// TIA Portal V16 program export: 10 tag tables, 22 data types, 19 data blocks, 13 code blocks (in call order from the OBs), 5 instance data blocks

VAR_GLOBAL   // PLC tag table "Default tag table"
END_VAR

VAR_GLOBAL   // PLC tag table "FC11001_Test"
   V001_FBK_OPEN AT %M100.0 : Bool;   // V001 Open limit switch
   V001_FBK_CLOSED AT %M100.1 : Bool;   // V001 Closed limit switch
   V001_FAULT AT %M100.2 : Bool;   // V001 External fault signal
   V001_OPERATE AT %M101.0 : Bool;   // V001 Energise (operate) signal
   V001_ESTOP AT %M100.3 : Bool;   // V001 Safety signal
   V001_TRIP AT %M100.4 : Bool;   // V001 Trip (interlock) signal
   V001_ILOCK AT %M100.5 : Bool;   // V001 Interlock signal
   V001_PERM AT %M100.6 : Bool;   // V001 Permissive (interlock) signal
   OpTimeRem AT %MD110 : Real;   // Operating timer last non-zero value
END_VAR

VAR_GLOBAL   // PLC tag table "FC19511_Test"
   SIM001_TRIGGER AT %M900.0 : Bool;   // Simulation Trigger Signal
   SIM001_OUTPUT AT %MD910 : Real;   // Simulation Output
   SIM001_INPUT AT %MD902 : Real;   // Simulation Input
   SIM001_Type AT %MW906 : Int;   // 0 = Step, 1 = Ramp, 2 = Sinusoid
   "Counter" AT %MW908 : Int;   // 100ms Counter
END_VAR

VAR_GLOBAL   // PLC tag table "FC19512"
   SIM001_TRIGGER AT %M900.0 : Bool;   // Simulation Trigger Signal
   SIM001_OUTPUT AT %MD910 : Real;
   SIM001_INPUT AT %MD902 : Real;
END_VAR

VAR_GLOBAL   // PLC tag table "PAL_FC11011_Test"
   V001_FBK_ENG AT %M100.0 : Bool;   // V001 Energised position limit switch
   V001_FBK_DENG AT %M100.1 : Bool;   // V001 Deenergised position limit switch
   V001_FAULT AT %M100.2 : Bool;   // V001 External fault signal
   V001_OPERATE AT %M101.0 : Bool;   // V001 Energise (operate) signal
   V001_ESTOP AT %M100.3 : Bool;   // V001 Safety signal
   V001_TRIP AT %M100.4 : Bool;   // V001 Trip (interlock) signal
   V001_ILOCK AT %M100.5 : Bool;   // V001 Interlock signal
   V001_PERM AT %M100.6 : Bool;   // V001 Permissive (interlock) signal
   OpTimeRem AT %MD110 : Real;   // Operating timer last non-zero value
END_VAR

VAR_GLOBAL   // PLC tag table "PAL_SystemTags"
   _SysSignals01 AT %MB0 : Byte;   // System signals byte 01 — Logic and scan synchronised pulses   {ExternalWritable false}
   _False AT %M0.0 : Bool;   // System Logic Bit — Always FALSE   {ExternalWritable false}
   _True AT %M0.1 : Bool;   // System Logic Bit — Always TRUE   {ExternalWritable false}
   _50ms AT %M0.2 : Bool;   // System Timing — 50 ms pulse scan synchronised   {ExternalWritable false}
   _100ms AT %M0.3 : Bool;   // System Timing — 100 ms pulse scan synchronised   {ExternalWritable false}
   _200ms AT %M0.4 : Bool;   // System Timing — 200 ms pulse scan synchronised   {ExternalWritable false}
   _500ms AT %M0.5 : Bool;   // System Timing — 500 ms pulse scan synchronised   {ExternalWritable false}
   _1s AT %M0.6 : Bool;   // System Timing — 1 s pulse scan synchronised   {ExternalWritable false}
   _2s AT %M0.7 : Bool;   // System Timing — 2 s pulse scan synchronised   {ExternalWritable false}
   _SysSignals02 AT %MB1 : Byte;   // System signals byte 02 — scan signals and common square waves   {ExternalWritable false}
   _CycleTick AT %M1.0 : Bool;   // System Timing — Cycle tick (active odd cycles, alternates with _CycleTock)   {ExternalWritable false}
   _CycleTock AT %M1.1 : Bool;   // System Timing — Cycle tock (active even cycles, alternates with _CycleTick)   {ExternalWritable false}
   _CycleFirst AT %M1.2 : Bool;   // System Timing — First cycle detected   {ExternalWritable false}
   _100msSqW AT %M1.3 : Bool;   // System Timing — 100 ms square wave scan synchronised   {ExternalWritable false}
   _200msSqW AT %M1.4 : Bool;   // System Timing — 200 ms square wave scan synchronised   {ExternalWritable false}
   _500msSqW AT %M1.5 : Bool;   // System Timing — 500 ms square wave scan synchronised   {ExternalWritable false}
   _1sSqW AT %M1.6 : Bool;   // System Timing — 1 s square wave scan synchronised   {ExternalWritable false}
   _2sSqW AT %M1.7 : Bool;   // System Timing — 2 s square wave scan synchronised   {ExternalWritable false}
   _ClockMem AT %MB10 : Byte;   // Clock Memory (populated by the CPU)   {ExternalWritable false}
   _ClockMem_100msSqW AT %M10.0 : Bool;   // Clock Memory — 10.0 Hz square wave 0.1 s period   {ExternalWritable false}
   _ClockMem_200msSqW AT %M10.1 : Bool;   // Clock Memory — 5.00 Hz square wave 0.2 s period   {ExternalWritable false}
   _ClockMem_400msSqW AT %M10.2 : Bool;   // Clock Memory — 2.50 Hz square wave 0.4 s period   {ExternalWritable false}
   _ClockMem_500msSqW AT %M10.3 : Bool;   // Clock Memory — 2.00 Hz square wave 0.5 s period   {ExternalWritable false}
   _ClockMem_800msSqW AT %M10.4 : Bool;   // Clock Memory — 1.25 Hz square wave 0.8 s period   {ExternalWritable false}
   _ClockMem_1000msSqW AT %M10.5 : Bool;   // Clock Memory — 1.00 Hz square wave 1.0 s period   {ExternalWritable false}
   _ClockMem_1600msSqW AT %M10.6 : Bool;   // Clock Memory — 0.62 Hz square wave 1.6 s period   {ExternalWritable false}
   _ClockMem_2000msSqW AT %M10.7 : Bool;   // Clock Memory — 0.50 Hz square wave 2.0 s period   {ExternalWritable false}
   _SysSignals AT %MW0 : Int;   // System signals   {ExternalWritable false}
END_VAR

VAR_GLOBAL   // PLC tag table "PAL_TestFC01001"
   Trap_dirFalseHigh AT %M12.0 : Bool;
   Trap_dirTrueLow AT %M12.1 : Bool;
   Trap_parFalseHigh AT %M12.2 : Bool;
   Trap_parTrueLow AT %M12.3 : Bool;
   Trap_dirCycFirstOn AT %M12.4 : Bool;
   Trap_parCycFirstOn AT %M12.5 : Bool;
   Trap_dirCycFirstCount AT %MW14 : Word;
   Trap_parCycFirstCount AT %MW16 : Word;
   Check_CycCount AT %MW1000 : Word;
END_VAR

VAR_GLOBAL   // PLC tag table "PAL_TestFC02001"
   FIC101_RAW AT %MW100 : Int;   // FIC101 - Instrument Simulation - RAW SIGNAL
   FIC101_FLT AT %M110.0 : Bool;   // FIC101 - Instrument Simulation - EXTERNAL FAULT
END_VAR

VAR_GLOBAL   // PLC tag table "PAL_TestFC18001"
   FIC101_RAW AT %MW100 : Int;   // FIC101 - Instrument Simulation - RAW SIGNAL
   OVER_RANGE AT %M102.0 : Bool;
   UNDER_RANGE AT %M102.1 : Bool;
   OUT_OF_RANGE AT %M102.2 : Bool;
   SCALE_VALUE AT %MD110 : Real;
END_VAR

VAR_GLOBAL   // PLC tag table "PAL_TestFC18151"
   EventTrigger AT %M20.0 : Bool;
END_VAR

TYPE "UT01000_St_SysRevision"
TITLE = Static UDT — Sys - Revision Data
// Revision Data
// stored: IsFailsafeCompliant false
   STRUCT
      REV_BLOCK { ExternalWritable := 'False'; S7_SetPoint := 'True'} : String[7];   // Block or Project number
      REV_NUMBER { ExternalWritable := 'False'; S7_SetPoint := 'True'} : String[20];   // Revision status followed by revision number
      REV_DATE { ExternalWritable := 'False'; S7_SetPoint := 'True'} : String[10];   // Revision date
      REV_AUTHOR { ExternalWritable := 'False'; S7_SetPoint := 'True'} : String[20];   // Revision author
   END_STRUCT;
END_TYPE

TYPE "UT01001_St_SysLicence"
TITLE = Static UDT [SYSTEM] — Licence Information
// PRACTICAL SERIES AUTOMATION LIBRARY (PAL)   —   COPYRIGHT 2020 – M. GLEDHILL (MIT LICENCE)
//                   ———— ◆ ————
// FULL ONLINE DOCUMENTATION IS AVAILABLE AT: https://practicalseries.com/2001-pal/index.html
// stored: IsFailsafeCompliant false
   STRUCT
      LICENCE_TYPE { ExternalWritable := 'False'} : String[20];   // Licence information — type of licence
      COPYRIGHT { ExternalWritable := 'False'} : String[30];   // Licence information — copyright (year and name)
   END_STRUCT;
END_TYPE

TYPE "UT00800_St_K_AnData"
TITLE = Static UDT [CONSTANTS] — Analog Card Ranges, Types and Coefficients
// PRACTICAL SERIES AUTOMATION LIBRARY (PAL)   —   COPYRIGHT 2020 – M. GLEDHILL (MIT LICENCE)
//                   ———— ◆ ————
// FULL ONLINE DOCUMENTATION IS AVAILABLE AT: https://practicalseries.com/2001-pal/index.html
// stored: IsFailsafeCompliant false
   STRUCT
      revInfo { ExternalWritable := 'False'} : "UT01000_St_SysRevision";   // ▀▀▀▀ UDT CURRENT REVISION
      ___________0010_0 { ExternalAccessible := 'False'; ExternalVisible := 'False'; ExternalWritable := 'False'} : Bool;
      ___________0010_1 { ExternalAccessible := 'False'; ExternalVisible := 'False'; ExternalWritable := 'False'} : Bool;   // ▀▀▀▀ AIO SIGNAL CODE
      AIO_CODE : UInt := 16#0000;   // Instrument code (type, coefficient and range)
      ___________0020_0 { ExternalAccessible := 'False'; ExternalVisible := 'False'; ExternalWritable := 'False'} : Bool := false;
      ___________0010_2 { ExternalAccessible := 'False'; ExternalVisible := 'False'; ExternalWritable := 'False'} : Bool;   // ▀▀▀▀ AIO RANGE DATA
      RAW_MIN : Int := 0;   // Minimum value of the analog input range
      RAW_MAX : Int := 27648;   // Maximum value of the analog input range
      RAW_NAME : String[60] := 'User defined instrument type';   // Signal type name
      ___________0030_1 { ExternalAccessible := 'False'; ExternalVisible := 'False'; ExternalWritable := 'False'} : Bool;
      ___________0030_2 { ExternalAccessible := 'False'; ExternalVisible := 'False'; ExternalWritable := 'False'} : Bool;   // ▀▀▀▀ AIO CARD PARAMETERS
      PARAM_TYPE : Byte := 16#00;   // Unique measurement type code
      PARAM_RANGE : Byte := 16#00;   // Unique measurement range code
      PARAM_COEF : Byte := 16#00;   // Unique temperature coefficient code (thermal resistance only)
      VALUE_COEF : Real;   // Temperature coefficient actual value, Ω/Ω/°C (thermal resistance only)
   END_STRUCT;
   // revInfo.REV_BLOCK := 'UT00800';
   // revInfo.REV_NUMBER := '000.101';
   // revInfo.REV_DATE := '2024-04-09';
   // revInfo.REV_AUTHOR := 'M. Gledhill';
END_TYPE

TYPE "UT00800_St_ConstAiRawData"
TITLE = Static UDT [SYSTEM CONSTANTS] — Analog Input Card Types, Ranges and Coefficients
// PRACTICAL SERIES AUTOMATION LIBRARY (PAL)   —   COPYRIGHT 2020 – M. GLEDHILL (MIT LICENCE)
//                   ———— ◆ ————
// FULL ONLINE DOCUMENTATION IS AVAILABLE AT: https://practicalseries.com/2001-pal/index.html
// stored: IsFailsafeCompliant false
   STRUCT
      revInfo { ExternalWritable := 'False'} : "UT01000_St_SysRevision";   // ▀▀▀▀ UDT CURRENT REVISION
      ___________0010_0 { ExternalAccessible := 'False'; ExternalVisible := 'False'; ExternalWritable := 'False'} : Bool;
      ___________0010_1 { ExternalAccessible := 'False'; ExternalVisible := 'False'; ExternalWritable := 'False'} : Bool;   // ▀▀▀▀ AI SIGNAL CODE
      AI_CODE { ExternalWritable := 'False'} : UInt := 16#0000;   // Input code (type, coefficient and range)
      ___________0020_0 { ExternalAccessible := 'False'; ExternalVisible := 'False'; ExternalWritable := 'False'} : Bool := false;
      ___________0010_2 { ExternalAccessible := 'False'; ExternalVisible := 'False'; ExternalWritable := 'False'} : Bool;   // ▀▀▀▀ AI RANGE DATA
      RAW_MIN { ExternalWritable := 'False'} : Int := 0;   // Minimum value of the analog input range
      RAW_MAX { ExternalWritable := 'False'} : Int := 27648;   // Maximum value of the analog input range
      RAW_NAME { ExternalWritable := 'False'} : String[60] := 'User defined instrument type';   // Signal type name
      ___________0030_1 { ExternalAccessible := 'False'; ExternalVisible := 'False'; ExternalWritable := 'False'} : Bool;
      ___________0030_2 { ExternalAccessible := 'False'; ExternalVisible := 'False'; ExternalWritable := 'False'} : Bool;   // ▀▀▀▀ AI CARD PARAMETERS
      PARAM_TYPE { ExternalWritable := 'False'} : Byte := 16#00;   // Unique measurement type code
      PARAM_RANGE { ExternalWritable := 'False'} : Byte := 16#00;   // Unique measurement range code
      PARAM_COEF { ExternalWritable := 'False'} : Byte := 16#00;   // Unique temperature coefficient code (thermal resistance only)
      ___________0040_1 { ExternalAccessible := 'False'; ExternalVisible := 'False'; ExternalWritable := 'False'} : Bool;
      ___________0040_2 { ExternalAccessible := 'False'; ExternalVisible := 'False'; ExternalWritable := 'False'} : Bool;   // ▀▀▀▀ AI CARD COEFFICIENTS
      VALUE_COEF { ExternalWritable := 'False'} : Real;   // Temperature coefficient actual value, Ω/Ω/°C (thermal resistance only)
   END_STRUCT;
   // revInfo.REV_BLOCK := 'UT00800';
   // revInfo.REV_NUMBER := '001.000';
   // revInfo.REV_DATE := '2024-04-09';
   // revInfo.REV_AUTHOR := 'M. Gledhill';
END_TYPE

TYPE "UT00801_St_ConstAiRawData"
TITLE = Static UDT [SYSTEM CONSTANTS] — Analog Input Card Types, Ranges and Coefficients
// PRACTICAL SERIES AUTOMATION LIBRARY (PAL)   —   COPYRIGHT 2020 – M. GLEDHILL (MIT LICENCE)
//                   ———— ◆ ————
// FULL ONLINE DOCUMENTATION IS AVAILABLE AT: https://practicalseries.com/2001-pal/index.html
// stored: IsFailsafeCompliant false
   STRUCT
      revInfo { ExternalWritable := 'False'} : "UT01000_St_SysRevision";   // ▀▀▀▀ UDT CURRENT REVISION
      ___________0010_0 { ExternalAccessible := 'False'; ExternalVisible := 'False'; ExternalWritable := 'False'} : Bool;
      ___________0010_1 { ExternalAccessible := 'False'; ExternalVisible := 'False'; ExternalWritable := 'False'} : Bool;   // ▀▀▀▀ AI SIGNAL CODE
      AI_CODE { ExternalWritable := 'False'} : UInt := 16#0000;   // Input code (type, coefficient and range)
      ___________0020_0 { ExternalAccessible := 'False'; ExternalVisible := 'False'; ExternalWritable := 'False'} : Bool := false;
      ___________0020_1 { ExternalAccessible := 'False'; ExternalVisible := 'False'; ExternalWritable := 'False'} : Bool;   // ▀▀▀▀ AI RANGE DATA
      RAW_MIN { ExternalWritable := 'False'} : Int := 0;   // Minimum value of the analog input range
      RAW_MAX { ExternalWritable := 'False'} : Int := 27648;   // Maximum value of the analog input range
      RAW_DESC { ExternalWritable := 'False'} : String[60] := 'User defined instrument type';   // Signal type description (plain English)
      ___________0030_1 { ExternalAccessible := 'False'; ExternalVisible := 'False'; ExternalWritable := 'False'} : Bool;
      ___________0030_2 { ExternalAccessible := 'False'; ExternalVisible := 'False'; ExternalWritable := 'False'} : Bool;   // ▀▀▀▀ AI CARD PARAMETERS
      PARAM_TYPE { ExternalWritable := 'False'} : Byte := 16#00;   // Unique measurement type code
      PARAM_RANGE { ExternalWritable := 'False'} : Byte := 16#00;   // Unique measurement range code
      PARAM_COEF { ExternalWritable := 'False'} : Byte := 16#00;   // Unique temperature coefficient code (thermal resistance only)
      ___________0040_1 { ExternalAccessible := 'False'; ExternalVisible := 'False'; ExternalWritable := 'False'} : Bool;
      ___________0040_2 { ExternalAccessible := 'False'; ExternalVisible := 'False'; ExternalWritable := 'False'} : Bool;   // ▀▀▀▀ AI CARD COEFFICIENTS
      VALUE_COEF { ExternalWritable := 'False'} : Real;   // Temperature coefficient actual value, Ω/Ω/°C (thermal resistance only)
   END_STRUCT;
   // revInfo.REV_BLOCK := 'UT00801';
   // revInfo.REV_NUMBER := '001.000';
   // revInfo.REV_DATE := '2024-04-09';
   // revInfo.REV_AUTHOR := 'M. Gledhill';
END_TYPE

TYPE "UT00802_St_ConstAqRawData"
TITLE = Static UDT [SYSTEM CONSTANTS] — Analog Input Card Types, Ranges and Coefficients
// PRACTICAL SERIES AUTOMATION LIBRARY (PAL)   —   COPYRIGHT 2020 – M. GLEDHILL (MIT LICENCE)
//                   ———— ◆ ————
// FULL ONLINE DOCUMENTATION IS AVAILABLE AT: https://practicalseries.com/2001-pal/index.html
// stored: IsFailsafeCompliant false
   STRUCT
      revInfo { ExternalWritable := 'False'} : "UT01000_St_SysRevision";   // ▀▀▀▀ UDT CURRENT REVISION
      ___________0010_0 { ExternalAccessible := 'False'; ExternalVisible := 'False'; ExternalWritable := 'False'} : Bool;
      ___________0010_1 { ExternalAccessible := 'False'; ExternalVisible := 'False'; ExternalWritable := 'False'} : Bool;   // ▀▀▀▀ AQ SIGNAL CODE
      AQ_CODE { ExternalWritable := 'False'} : UInt := 16#0000;   // Input code (type, coefficient and range)
      ___________0020_0 { ExternalAccessible := 'False'; ExternalVisible := 'False'; ExternalWritable := 'False'} : Bool := false;
      ___________0020_1 { ExternalAccessible := 'False'; ExternalVisible := 'False'; ExternalWritable := 'False'} : Bool;   // ▀▀▀▀ AQ RANGE DATA
      RAW_MIN { ExternalWritable := 'False'} : Int := 0;   // Minimum value of the analog input range
      RAW_MAX { ExternalWritable := 'False'} : Int := 27648;   // Maximum value of the analog input range
      RAW_DESC { ExternalWritable := 'False'} : String[60] := 'User defined instrument type';   // Signal type description (plain English)
      ___________0030_1 { ExternalAccessible := 'False'; ExternalVisible := 'False'; ExternalWritable := 'False'} : Bool;
      ___________0030_2 { ExternalAccessible := 'False'; ExternalVisible := 'False'; ExternalWritable := 'False'} : Bool;   // ▀▀▀▀ AQ CARD PARAMETERS
      PARAM_TYPE { ExternalWritable := 'False'} : Byte := 16#00;   // Unique measurement type code
      PARAM_RANGE { ExternalWritable := 'False'} : Byte := 16#00;   // Unique measurement range code
   END_STRUCT;
   // revInfo.REV_BLOCK := 'UT00802';
   // revInfo.REV_NUMBER := '001.000';
   // revInfo.REV_DATE := '2024-05-16';
   // revInfo.REV_AUTHOR := 'M. Gledhill';
END_TYPE

TYPE "UT00851_Sy_ConstAiScaleData"
TITLE = Static UDT [SYSTEM CONSTANTS] — Analog Input Scale Data and Ranges
// PRACTICAL SERIES AUTOMATION LIBRARY (PAL)   —   COPYRIGHT 2020 – M. GLEDHILL (MIT LICENCE)
//                   ———— ◆ ————
// FULL ONLINE DOCUMENTATION IS AVAILABLE AT: https://practicalseries.com/2001-pal/index.html
// stored: IsFailsafeCompliant false
   STRUCT
      revInfo { ExternalWritable := 'False'} : "UT01000_St_SysRevision";   // ▀▀▀▀ UDT CURRENT REVISION
      ___________0010_0 { ExternalAccessible := 'False'; ExternalVisible := 'False'; ExternalWritable := 'False'} : Bool;
      ___________0010_1 { ExternalAccessible := 'False'; ExternalVisible := 'False'; ExternalWritable := 'False'} : Bool;   // ▀▀▀▀ AI DEVICE ID
      AI_TAG { ExternalWritable := 'False'} : String[20] := 'AAAnnn';   // Device or instrument tag
      ___________0020_0 { ExternalAccessible := 'False'; ExternalVisible := 'False'; ExternalWritable := 'False'} : Bool := false;
      ___________0020_1 { ExternalAccessible := 'False'; ExternalVisible := 'False'; ExternalWritable := 'False'} : Bool;   // ▀▀▀▀ AI SCALED RANGE DATA
      SCALE_MIN { ExternalWritable := 'False'} : Real := 0.0;   // Minimum value of the scaled signal
      SCALE_MAX { ExternalWritable := 'False'} : Real := 100.0;   // Maximum value of the scaled signal
      SCALE_UNITS { ExternalWritable := 'False'} : String[20] := '%';   // Scaled signal engineering units
      SCALE_DESC { ExternalWritable := 'False'} : String[60] := 'Default range 0.0-100.0%';   // Scaled signal type information (plain English)
      ___________0030_0 { ExternalAccessible := 'False'; ExternalVisible := 'False'; ExternalWritable := 'False'} : Bool := false;
      ___________0030_1 { ExternalAccessible := 'False'; ExternalVisible := 'False'; ExternalWritable := 'False'} : Bool;   // ▀▀▀▀ AI OUT OF RANGE DATA
      LIMIT_UNDER { ExternalWritable := 'False'} : Real := 0.0;   // Lower limit of scaled signal before under-range (in engineering uints)
      LIMIT_OVER { ExternalWritable := 'False'} : Real := 100.0;   // Upper limit of scaled signal before over-range (in engineering uints)
      ___________0040_0 { ExternalAccessible := 'False'; ExternalVisible := 'False'; ExternalWritable := 'False'} : Bool := false;
      ___________0040_1 { ExternalAccessible := 'False'; ExternalVisible := 'False'; ExternalWritable := 'False'} : Bool;   // ▀▀▀▀ AI USER INFORMATION
      USER_INFO_1 : String[60] := 'Optional user information';   // Optional user information (text) line 1
      USER_INFO_2 : String[60] := 'Optional user information';   // Optional user information (text) line 2
      USER_INFO_3 : String[60] := 'Optional user information';   // Optional user information (text) line 3
      USER_INFO_4 : String[60] := 'Optional user information';   // Optional user information (text) line 4
      USER_INFO_5 : String[60] := 'Optional user information';   // Optional user information (text) line 5
   END_STRUCT;
   // revInfo.REV_BLOCK := 'UT00851';
   // revInfo.REV_NUMBER := '001.000';
   // revInfo.REV_DATE := '2024-05-11';
   // revInfo.REV_AUTHOR := 'M. Gledhill';
END_TYPE

TYPE "UT00852_Sy_ConstAqScaleData"
TITLE = Static UDT [SYSTEM CONSTANTS] — Analog Input Scale Data and Ranges
// PRACTICAL SERIES AUTOMATION LIBRARY (PAL)   —   COPYRIGHT 2020 – M. GLEDHILL (MIT LICENCE)
//                   ———— ◆ ————
// FULL ONLINE DOCUMENTATION IS AVAILABLE AT: https://practicalseries.com/2001-pal/index.html
// stored: IsFailsafeCompliant false
   STRUCT
      revInfo { ExternalWritable := 'False'} : "UT01000_St_SysRevision";   // ▀▀▀▀ UDT CURRENT REVISION
      ___________0010_0 { ExternalAccessible := 'False'; ExternalVisible := 'False'; ExternalWritable := 'False'} : Bool;
      ___________0010_1 { ExternalAccessible := 'False'; ExternalVisible := 'False'; ExternalWritable := 'False'} : Bool;   // ▀▀▀▀ AQ DEVICE ID
      AQ_TAG { ExternalWritable := 'False'} : String[20] := 'AAAnnn';   // Device tag
      ___________0020_0 { ExternalAccessible := 'False'; ExternalVisible := 'False'; ExternalWritable := 'False'} : Bool := false;
      ___________0020_1 { ExternalAccessible := 'False'; ExternalVisible := 'False'; ExternalWritable := 'False'} : Bool;   // ▀▀▀▀ AQ SCALED RANGE DATA
      SCALE_MIN { ExternalWritable := 'False'} : Real := 0.0;   // Minimum value of the scaled signal
      SCALE_MAX { ExternalWritable := 'False'} : Real := 100.0;   // Maximum value of the scaled signal
      SCALE_UNITS { ExternalWritable := 'False'} : String[20] := '%';   // Scaled signal engineering units
      SCALE_DESC { ExternalWritable := 'False'} : String[60] := 'Default range 0.0-100.0%';   // Scaled signal type description (plain English)
      ___________0030_0 { ExternalAccessible := 'False'; ExternalVisible := 'False'; ExternalWritable := 'False'} : Bool := false;
      ___________0030_1 { ExternalAccessible := 'False'; ExternalVisible := 'False'; ExternalWritable := 'False'} : Bool;   // ▀▀▀▀ AQ OUT OF RANGE DATA
      LIMIT_UNDER { ExternalWritable := 'False'} : Real := 0.0;   // Lower limit of scaled signal before under-range (in engineering uints)
      LIMIT_OVER { ExternalWritable := 'False'} : Real := 100.0;   // Upper limit of scaled signal before over-range (in engineering uints)
      ___________0040_0 { ExternalAccessible := 'False'; ExternalVisible := 'False'; ExternalWritable := 'False'} : Bool := false;
      ___________0040_1 { ExternalAccessible := 'False'; ExternalVisible := 'False'; ExternalWritable := 'False'} : Bool;   // ▀▀▀▀ AQ USER INFORMATION
      USER_INFO_1 : String[60] := 'Optional user information';   // Optional user information (text) line 1
      USER_INFO_2 : String[60] := 'Optional user information';   // Optional user information (text) line 2
      USER_INFO_3 : String[60] := 'Optional user information';   // Optional user information (text) line 3
      USER_INFO_4 : String[60] := 'Optional user information';   // Optional user information (text) line 4
      USER_INFO_5 : String[60] := 'Optional user information';   // Optional user information (text) line 5
   END_STRUCT;
   // revInfo.REV_BLOCK := 'UT00852';
   // revInfo.REV_NUMBER := '001.000';
   // revInfo.REV_DATE := '2024-05-16';
   // revInfo.REV_AUTHOR := 'M. Gledhill';
END_TYPE

TYPE "UT21000_Dy_SysSignals"
TITLE = Dynamic UDT — Sys - Global Signals
// Global Logic and Timing Signals
// stored: IsFailsafeCompliant false
   STRUCT
      revInfo { ExternalWritable := 'False'} : "UT01000_St_SysRevision";   // ▀▀▀▀ UDT CURRENT REVISION
      ___________0010_0 { ExternalAccessible := 'False'; ExternalVisible := 'False'; ExternalWritable := 'False'} : Bool;
      ___________0010_1 { ExternalAccessible := 'False'; ExternalVisible := 'False'; ExternalWritable := 'False'} : Bool;   // ▀▀▀▀ SYSTEM SIGNALS
      _False { ExternalWritable := 'False'} : Bool;   // System Logic Bit — Always FALSE
      _True { ExternalWritable := 'False'} : Bool;   // System Logic Bit — Always TRUE
      _50ms { ExternalWritable := 'False'} : Bool;   // System Timing — 50 ms Pulse Scan synchronised
      _100ms { ExternalWritable := 'False'} : Bool;   // System Timing — 100 ms Pulse Scan synchronised
      _200ms { ExternalWritable := 'False'} : Bool;   // System Timing — 200 ms Pulse Scan synchronised
      _500ms { ExternalWritable := 'False'} : Bool;   // System Timing — 500 ms Pulse Scan synchronised
      _1s { ExternalWritable := 'False'} : Bool;   // System Timing — 1 s Pulse Scan synchronised
      _2s { ExternalWritable := 'False'} : Bool;   // System Timing — 2 s Pulse Scan synchronised
      _CycleTick { ExternalWritable := 'False'} : Bool;   // System Timing — Cycle tick (active odd cycles, alternates with _CycleTock)
      _CycleTock { ExternalWritable := 'False'} : Bool;   // System Timing — Cycle tock (active even cycles, alternates with _CycleTick)
      _CycleFirst { ExternalWritable := 'False'} : Bool;   // System Timing — First cycle detected
      _100msSqW { ExternalWritable := 'False'} : Bool;   // System Timing — 100 ms Square wave Scan synchronised
      _200msSqW { ExternalWritable := 'False'} : Bool;   // System Timing — 200 ms Square wave Scan synchronised
      _500msSqW { ExternalWritable := 'False'} : Bool;   // System Timing — 500 ms Square wave Scan synchronised
      _1sSqW { ExternalWritable := 'False'} : Bool;   // System Timing — 1 s Square wave Scan synchronised
      _2sSqW { ExternalWritable := 'False'} : Bool;   // System Timing — 2 s Square wave Scan synchronised
   END_STRUCT;
   // revInfo.REV_BLOCK := 'UT21000';
   // revInfo.REV_NUMBER := '000.801';
   // revInfo.REV_DATE := '2021-05-11';
   // revInfo.REV_AUTHOR := 'M. Gledhill';
END_TYPE

TYPE "UT21001_Dy_SysData"
TITLE = Dynamic UDT [SYSTEM] — Global Data
// PRACTICAL SERIES AUTOMATION LIBRARY (PAL)   —   COPYRIGHT 2020 – M. GLEDHILL (MIT LICENCE)
//                   ———— ◆ ————
// FULL ONLINE DOCUMENTATION IS AVAILABLE AT: https://practicalseries.com/2001-pal/index.html
// stored: IsFailsafeCompliant false
   STRUCT
      revInfo { ExternalWritable := 'False'} : "UT01000_St_SysRevision";   // ▀▀▀▀ UDT CURRENT REVISION
      ___________0010_0 { ExternalAccessible := 'False'; ExternalVisible := 'False'; ExternalWritable := 'False'} : Bool;
      ___________0010_1 { ExternalAccessible := 'False'; ExternalVisible := 'False'; ExternalWritable := 'False'} : Bool;   // ▀▀▀▀ CYCLE TIME DATA
      CycTime_Prev { ExternalWritable := 'False'} : Real;   // Previous cycle time (ms)
      CycTime_Max { ExternalWritable := 'False'} : Real;   // Maximum cycle time - since start-up (ms)
      CycTime_Min { ExternalWritable := 'False'} : Real;   // Minimum cycle time - since start-up (ms)
      Cyc_Counter { ExternalWritable := 'False'} : UDInt;   // Cycle rolling counter - incremented by 1 each scan
      __________0020_0 { ExternalAccessible := 'False'; ExternalVisible := 'False'; ExternalWritable := 'False'} : Bool := false;
      __________0020_1 { ExternalAccessible := 'False'; ExternalVisible := 'False'; ExternalWritable := 'False'} : Bool := false;   // ▀▀▀▀ REAL TIME CLOCK DATA
      RTC_Year { ExternalWritable := 'False'} : Int;   // Year (returns a value in the range 1970 to 2262)
      RTC_Month { ExternalWritable := 'False'} : Int;   // Month (1-12 representing Jan to Dec)
      RTC_Day { ExternalWritable := 'False'} : Int;   // Day of month (1-31)
      RTC_DayofWeek { ExternalWritable := 'False'} : Int;   // Day of week (1-7, where 1=Sunday, 7=Saturday)
      RTC_Hour { ExternalWritable := 'False'} : Int;   // Hour of day (0-23)
      RTC_Minute { ExternalWritable := 'False'} : Int;   // Minutes (0-59)
      RTC_Second { ExternalWritable := 'False'} : Int;   // Seconds (0-59)
      RTC_millisecond { ExternalWritable := 'False'} : Int;   // Milliseconds (0-999)
   END_STRUCT;
   // revInfo.REV_BLOCK := 'UT21001';
   // revInfo.REV_NUMBER := '001.102';
   // revInfo.REV_DATE := '2022-04-04';
   // revInfo.REV_AUTHOR := 'M. Gledhill';
END_TYPE

TYPE "UT02001_St_InstAnalogRead"
TITLE = Static UDT [INSTRUMENTATION] — Analog Instrument Read, Scale and Monitor
// PRACTICAL SERIES AUTOMATION LIBRARY (PAL)   —   COPYRIGHT 2020 – M. GLEDHILL (MIT LICENCE)
//                   ———— ◆ ————
// FULL ONLINE DOCUMENTATION IS AVAILABLE AT: https://practicalseries.com/2001-pal/index.html
// stored: IsFailsafeCompliant false
   STRUCT
      revInfo { ExternalWritable := 'False'} : "UT01000_St_SysRevision";   // Revision information
      ___________0010_0 { ExternalAccessible := 'False'; ExternalVisible := 'False'; ExternalWritable := 'False'} : Int;
      ___________0010_1 { ExternalAccessible := 'False'; ExternalVisible := 'False'; ExternalWritable := 'False'} : Int;   // ▀▀▀▀ INSTRUMENT CONFIGURATION
      CONFIG_ALM_H_EN { ExternalWritable := 'False'; S7_SetPoint := 'True'} : Bool;   // CONFIG — High alarm is enabled (1 = enabled, 0 = no alarm)
      CONFIG_ALM_L_EN { ExternalWritable := 'False'; S7_SetPoint := 'True'} : Bool;   // CONFIG — Low alarm is enabled (1 = enabled, 0 = no alarm)
      CONFIG_WRN_H_EN { ExternalWritable := 'False'; S7_SetPoint := 'True'} : Bool;   // CONFIG — High warning is enabled (1 = enabled, 0 = no warning)
      CONFIG_WRN_L_EN { ExternalWritable := 'False'; S7_SetPoint := 'True'} : Bool;   // CONFIG — Low warning is enabled (1 = enabled, 0 = no warning)
      CONFIG_FP_DIS { ExternalWritable := 'False'; S7_SetPoint := 'True'} : Bool := false;   // CONFIG — Faceplate is disabled (1 = no Faceplate, 0 = normal)
      CONFIG_SIM_DIS { ExternalWritable := 'False'; S7_SetPoint := 'True'} : Bool := false;   // CONFIG — Simulation mode is disabled (1 = no Simulation, 0 = normal)
      CONFIG_RL_EN { ExternalWritable := 'False'; S7_SetPoint := 'True'} : Bool := false;   // CONFIG — Remote/local mode enabled (1 = remote/local permitted, 0 = remote/local N/A)
      ___________0020_0 { ExternalAccessible := 'False'; ExternalVisible := 'False'; ExternalWritable := 'False'} : Int;
      ___________0020_1 { ExternalAccessible := 'False'; ExternalVisible := 'False'; ExternalWritable := 'False'} : Int;   // ▀▀▀▀ INSTRUMENT RANGE & SCALING DATA
      RANGE_RAW_MIN { ExternalWritable := 'False'; S7_SetPoint := 'True'} : Int;   // RANGE — Minimum value of the raw analog signal (at the card)
      RANGE_RAW_MAX { ExternalWritable := 'False'; S7_SetPoint := 'True'} : Int;   // RANGE — Maximum value of the raw analog signal (at the card)
      RANGE_SCALE_MIN { ExternalWritable := 'False'; S7_SetPoint := 'True'} : Real;   // RANGE — Minimum value of the scaled analog signal [engineering units]
      RANGE_SCALE_MAX { ExternalWritable := 'False'; S7_SetPoint := 'True'} : Real;   // RANGE — Maximum value of the scaled analog signal [engineering units]
      RANGE_OOR_PERCENT { ExternalWritable := 'False'; S7_SetPoint := 'True'} : Real;   // RANGE — Out of range percentage (of raw range), beyond which the instrument is out of range
      ___________0030_0 { ExternalAccessible := 'False'; ExternalVisible := 'False'; ExternalWritable := 'False'} : Int;
      ___________0030_1 { ExternalAccessible := 'False'; ExternalVisible := 'False'; ExternalWritable := 'False'} : Int;   // ▀▀▀▀ INSTRUMENT INFORMATION (TAG & UNITS)
      INFO_TYPE : Int;   // INFORMATION — Instrument type (000 voltage, 100 current, 200 RTD 300 Thermocouple)
      INFO_TAG { ExternalWritable := 'False'; S7_SetPoint := 'True'} : String[20];   // INFORMATION — Instrument ID tag
      INFO_UNITS { ExternalWritable := 'False'; S7_SetPoint := 'True'} : String[10];   // INFORMATION — Engineering units of the instrument (unit of measure)
      ___________0040_0 { ExternalAccessible := 'False'; ExternalVisible := 'False'; ExternalWritable := 'False'} : Int;
      ___________0040_1 { ExternalAccessible := 'False'; ExternalVisible := 'False'; ExternalWritable := 'False'} : Int;   // ▀▀▀▀ INSTRUMENT ALARM/WARNING & HYSTERESIS SETPOINTS
      SP_ALM_H_VAL { ExternalWritable := 'False'; S7_SetPoint := 'True'} : Real;   // SETPOINT — High alarm threshold value [engineering units]
      SP_ALM_L_VAL { ExternalWritable := 'False'; S7_SetPoint := 'True'} : Real;   // SETPOINT — Low alarm threshold value [engineering units]
      SP_WRN_H_VAL { ExternalWritable := 'False'; S7_SetPoint := 'True'} : Real;   // SETPOINT — High warning threshold value [engineering units]
      SP_WRN_L_VAL { ExternalWritable := 'False'; S7_SetPoint := 'True'} : Real;   // SETPOINT — Low warning threshold value [engineering units]
      SP_ALM_H_HYST_VAL { ExternalWritable := 'False'; S7_SetPoint := 'True'} : Real;   // SETPOINT — High alarm hysteresis value [engineering units]
      SP_ALM_L_HYST_VAL { ExternalWritable := 'False'; S7_SetPoint := 'True'} : Real;   // SETPOINT — Low alarm hysteresis value [engineering units]
      SP_WRN_H_HYST_VAL { ExternalWritable := 'False'; S7_SetPoint := 'True'} : Real;   // SETPOINT — High warning hysteresis value [engineering units]
      SP_WRN_L_HYST_VAL { ExternalWritable := 'False'; S7_SetPoint := 'True'} : Real;   // SETPOINT — Low warning hysteresis value [engineering units]
      ___________0050_0 { ExternalAccessible := 'False'; ExternalVisible := 'False'; ExternalWritable := 'False'} : Int;
      ___________0050_1 { ExternalAccessible := 'False'; ExternalVisible := 'False'; ExternalWritable := 'False'} : Int;   // ▀▀▀▀ INSTRUMENT TIMER DEFAULT VALUES
      TIME_ALM_H_ON_DEL { ExternalWritable := 'False'; S7_SetPoint := 'True'} : Real;   // TIMER — High alarm on delay time (activation delay), [seconds]
      TIME_ALM_L_ON_DEL { ExternalWritable := 'False'; S7_SetPoint := 'True'} : Real;   // TIMER — Low alarm on delay time (activation delay), [seconds]
      TIME_WRN_H_ON_DEL { ExternalWritable := 'False'; S7_SetPoint := 'True'} : Real;   // TIMER — High warning on delay time (activation delay), [seconds]
      TIME_WRN_L_ON_DEL { ExternalWritable := 'False'; S7_SetPoint := 'True'} : Real;   // TIMER — Low warning on delay time (activation delay), [seconds]
      TIME_ALM_H_OFF_DEL { ExternalWritable := 'False'; S7_SetPoint := 'True'} : Real;   // TIMER — High alarm off delay time (deactivation delay), [seconds]
      TIME_ALM_L_OFF_DEL { ExternalWritable := 'False'; S7_SetPoint := 'True'} : Real;   // TIMER — Low alarm off delay time (deactivation delay), [seconds]
      TIME_WRN_H_OFF_DEL { ExternalWritable := 'False'; S7_SetPoint := 'True'} : Real;   // TIMER — High warning off delay time (deactivation delay), [seconds]
      TIME_WRN_L_OFF_DEL { ExternalWritable := 'False'; S7_SetPoint := 'True'} : Real;   // TIMER — Low warning off delay time (deactivation delay), [seconds]
   END_STRUCT;
   // revInfo.REV_BLOCK := 'UT02001';
   // revInfo.REV_NUMBER := '001.801';
   // revInfo.REV_DATE := '2022-04-11';
   // revInfo.REV_AUTHOR := 'M. Gledhill';
END_TYPE

TYPE "UT22001_Dy_InstAnalogRead"
TITLE = Dynamic UDT [INSTRUMENTATION] — Analog Instrument Read, Scale and Monitor
// PRACTICAL SERIES AUTOMATION LIBRARY (PAL)   —   COPYRIGHT 2020 – M. GLEDHILL (MIT LICENCE)
//                   ———— ◆ ————
// FULL ONLINE DOCUMENTATION IS AVAILABLE AT: https://practicalseries.com/2001-pal/index.html
// stored: IsFailsafeCompliant false
   STRUCT
      revInfo : "UT01000_St_SysRevision";   // Revision information
      ___________0010_0 { ExternalAccessible := 'False'; ExternalVisible := 'False'; ExternalWritable := 'False'} : Int;
      ___________0010_1 { ExternalAccessible := 'False'; ExternalVisible := 'False'; ExternalWritable := 'False'} : Int;   // ▀▀▀▀ STATUS (FOR BLOCK ICON AND SYMBOL)
      status_ConfigError : Bool;   // STATUS — Block is configured incorrectly
      status_Alm_H : Bool;   // STATUS — High alarm is active (1 = alarm active, 0 = no alarm)
      status_Alm_L : Bool;   // STATUS — Low alarm is active (1 = alarm active, 0 = no alarm)
      status_Wrn_H : Bool;   // STATUS — High warning is active (1 = warning active, 0 = no warning)
      status_Wrn_L : Bool;   // STATUS — Low warning is active (1 = warning active, 0 = no warning)
      status_Alm_H_Mask : Bool;   // STATUS — High alarm is masked (1 = alarm masked, 0 = normal)
      status_Alm_L_Mask : Bool;   // STATUS — Low alarm is masked (1 = alarm masked, 0 = normal)
      status_Wrn_H_Mask : Bool;   // STATUS — High warning is masked (1 = warning masked, 0 = normal)
      status_Wrn_L_Mask : Bool;   // STATUS — Low warning is masked (1 = warning masked, 0 = normal)
      status_Alm_H_Dis : Bool;   // STATUS — High alarm is disabled (1 = alarm disabled, 0 = normal)
      status_Alm_L_Dis : Bool;   // STATUS — Low alarm is disabled (1 = alarm disabled, 0 = normal)
      status_Wrn_H_Dis : Bool;   // STATUS — High warning is disabled (1 = warning disabled, 0 = normal)
      status_Wrn_L_Dis : Bool;   // STATUS — Low warning is disabled (1 = warning disabled, 0 = normal)
      status_Fault : Bool;   // STATUS — Device is in fault (1 = fault present, 0 = healthy)
      status_SimOn : Bool;   // STATUS — Device is in simulation mode (1 = simulation mode on, 0 = normal)
      status_RemoteOn : Bool;   // STATUS — Device is in remote mode (1 = remote mode, 0 = remote mode off)
      status_LocalOn : Bool;   // STATUS — Device is in local mode (1 = local mode, 0 = local mode off)
      status_RLOff : Bool;   // STATUS — Remote/local mode disabled (1 = ALL mode on, 0 = RL mode selected)
      ___________0020_0 { ExternalAccessible := 'False'; ExternalVisible := 'False'; ExternalWritable := 'False'} : Int;
      ___________0020_1 { ExternalAccessible := 'False'; ExternalVisible := 'False'; ExternalWritable := 'False'} : Int;   // ▀▀▀▀ CALCULATED VALUES (ABSOLUTE OVER AND UNDER RANGE)
      cal_OR_Abs : Real;   // CALC — Over-range limit (absolute value)
      cal_UR_Abs : Real;   // CALC — Under-range limit (absolute value)
      ___________0030_0 { ExternalAccessible := 'False'; ExternalVisible := 'False'; ExternalWritable := 'False'} : Int;
      ___________0030_2 { ExternalAccessible := 'False'; ExternalVisible := 'False'; ExternalWritable := 'False'} : Int;   // ▀▀▀▀ OPERATING MODE SELECTION (FROM FACEPLATE OR PANEL)
      mode_Alm_H_MaskOn : Bool;   // MODE — Mask Alm_H (1 = mask alarm, 0 = normal)
      mode_Alm_L_MaskOn : Bool;   // MODE — Mask Alm_L (1 = mask alarm, 0 = normal)
      mode_Wrn_H_MaskOn : Bool;   // MODE — Mask Wrn_H (1 = mask warning, 0 = normal)
      mode_Wrn_L_MaskOn : Bool;   // MODE — Mask Wrn_H (1 = mask warning, 0 = normal)
      mode_SimOn : Bool := false;   // MODE — Simulation mode (1 = simulation mode active, 0 = normal)
      mode_SimValue : Real;   // MODE — Simulation value [engineering units]
      mode_RemoteOn : Bool := false;   // MODE — Local HMI control enabled (1 = control active, 0 = control disabled or N/A)
      mode_LocalOn : Bool := false;   // MODE — Remote SCADA control enabled (1 = control active, 0 = control disabled or N/A)
      ___________0040_0 { ExternalAccessible := 'False'; ExternalVisible := 'False'; ExternalWritable := 'False'} : Int;
      ___________0040_1 { ExternalAccessible := 'False'; ExternalVisible := 'False'; ExternalWritable := 'False'} : Int;   // ▀▀▀▀ MESSAGES (ALARMS, WARNINGS, FAULTS AND EVENTS)
      msg_Alm_H : Bool;   // MESSAGE — Alarm - high alarm is active
      msg_Alm_L : Bool;   // MESSAGE — Alarm - low alarm is active
      msg_Wrn_H : Bool;   // MESSAGE — Warning - high warning is active
      msg_Wrn_L : Bool;   // MESSAGE — Warning - low warning is active
      msg_Flt_External : Bool;   // MESSAGE — Fault - external fault signal is active
      msg_Flt_OverRange : Bool;   // MESSAGE — Fault - instrument is over-range
      msg_Flt_UnderRange : Bool;   // MESSAGE — Fault - instrument is under-range
      msg_Flt_OutOfRange : Bool;   // MESSAGE — Fault - instrument is out-of-range
      ___________0050_0 { ExternalAccessible := 'False'; ExternalVisible := 'False'; ExternalWritable := 'False'} : Int;
      ___________0050_1 { ExternalAccessible := 'False'; ExternalVisible := 'False'; ExternalWritable := 'False'} : Int;   // ▀▀▀▀ BATCH AND BOOKING DATA
      batch_ID : UInt;   // BATCH — Booking ID (optional for batch operations)
      ___________0060_0 { ExternalAccessible := 'False'; ExternalVisible := 'False'; ExternalWritable := 'False'} : Int;
      ___________0060_1 { ExternalAccessible := 'False'; ExternalVisible := 'False'; ExternalWritable := 'False'} : Int;   // ▀▀▀▀ LIVE DATA (SCALED READING & TIMER VALUES)
      actual_Value : Real;   // ACTUAL — SCALED INSTRUMENT VALUE [engineering units]
      actual_Alm_H_Timer : Real;   // ACTUAL — Timer value — alarm high operation timer [seconds]
      actual_Alm_L_Timer : Real;   // ACTUAL — Timer value — alarm low operation timer [seconds]
      actual_Wrn_H_Timer : Real;   // ACTUAL — Timer value — warning high operation timer [seconds]
      actual_Wrn_L_Timer : Real;   // ACTUAL — Timer value — warning low operation timer [seconds]
      ___________0090_0 { ExternalAccessible := 'False'; ExternalVisible := 'False'; ExternalWritable := 'False'} : Int;
      ___________0090_1 { ExternalAccessible := 'False'; ExternalVisible := 'False'; ExternalWritable := 'False'} : Int;   // ▀▀▀▀ BLOCK INTERNAL WORKING AND STORAGE AREA
      "$pret_AlmHEn" : Bool;   // INTERNAL — Edge retention (+ve) alarm high enable
      "$Pret_AlmLEn" : Bool;   // INTERNAL — Edge retention (+ve) alarm low enable
      "$pret_WrnHEn" : Bool;   // INTERNAL — Edge retention (+ve) warning high enable
      "$pret_WrnLEn" : Bool;   // INTERNAL — Edge retention (+ve) warning low enable
   END_STRUCT;
   // revInfo.REV_BLOCK := 'UT22001';
   // revInfo.REV_NUMBER := '001.102';
   // revInfo.REV_DATE := '2022-04-08';
   // revInfo.REV_AUTHOR := 'M. Gledhill';
END_TYPE

TYPE "UT11001_St_DevValveIsol"
TITLE = Static UDT [Instrumentation] — Analog Instrument Read, Scale and Monitor
// Analogue Instrument Read and Scale
// stored: IsFailsafeCompliant false
   STRUCT
      revInfo { ExternalWritable := 'False'} : "UT01000_St_SysRevision";   // Revision information
      ___________0010_0 { ExternalAccessible := 'False'; ExternalVisible := 'False'; ExternalWritable := 'False'} : Int;
      ___________0010_1 { ExternalAccessible := 'False'; ExternalVisible := 'False'; ExternalWritable := 'False'} : Int;   // ▀▀▀▀ INSTRUMENT CONFIGURATION
      CONFIG_NO_NC : Bool;   // CONFIG — Normally open or normally closed valve (1 = normally open, 0 = normally closed)
      CONFIG_FBK_OPEN_EN : Bool;   // CONFIG — Open feedback is enabled (1 = open feedback present, 0 = no open feedback)
      CONFIG_FBK_CLOSED_EN : Bool;   // CONFIG — Closed feedback is enabled (1 = closed feedback present, 0 = no closed feedback)
      CONFIG_ESTOP_DIS : Bool;   // CONFIG — E_STOP signal disabled (1 = E_STOP not used, 0 = E_STOP in use)
      CONFIG_TRIP_DIS : Bool;   // CONFIG — TRIP signal disabled (1 = TRIP not used, 0 = TRIP in use)
      CONFIG_ILOCK_DIS : Bool;   // CONFIG — INTERLOCK signal disabled (1 = INTERLOCK not used, 0 = INTERLOCK in use)
      CONFIG_PERM_DIS : Bool;   // CONFIG — PERMISSIVE signal disabled (1 = PERMISSIVE not used, 0 = PERMISSIVE in use)
      CONFIG_TRIP_OP_CL : Bool;   // CONFIG — TRIP state (1 = open if tripped, 0 = close if tripped)
      CONFIG_ILOCK_OP_CL : Bool;   // CONFIG — INTERLOCK state (1 = open if interlocked, 0 = close if interlocked)
      CONFIG_PERM_OP_CL : Bool;   // CONFIG — PERMISSIVE permitted state (1 = permitted state open, 0 = permitted state closed)
      CONFIG_FP_DIS { ExternalWritable := 'False'; S7_SetPoint := 'True'} : Bool;   // CONFIG — Faceplate is disabled (1 = no Faceplate, 0 = normal)
      CONFIG_MAN_DIS : Bool;   // CONFIG — Manual mode is disabled (1 = no manual mode – auto only, 0 = normal)
      CONFIG_BYPASS_DIS : Bool;   // CONFIG — Bypass mode is disabled (1 = no Bypass, 0 = normal)
      CONFIG_SIM_DIS { ExternalWritable := 'False'; S7_SetPoint := 'True'} : Bool;   // CONFIG — Simulation mode is disabled (1 = no Simulation, 0 = normal)
      CONFIG_RL_EN { ExternalWritable := 'False'; S7_SetPoint := 'True'} : Bool;   // CONFIG — Remote/local mode enabled (1 = remote/local permitted, 0 = remote/local N/A)
      ___________0020_0 { ExternalAccessible := 'False'; ExternalVisible := 'False'; ExternalWritable := 'False'} : Int;
      ___________0020_1 { ExternalAccessible := 'False'; ExternalVisible := 'False'; ExternalWritable := 'False'} : Int;   // ▀▀▀▀ INSTRUMENT INFORMATION (TAG & UNITS)
      INFO_TAG { ExternalWritable := 'False'; S7_SetPoint := 'True'} : String[20];   // INFORMATION — Instrument ID tag
      ___________0030_0 { ExternalAccessible := 'False'; ExternalVisible := 'False'; ExternalWritable := 'False'} : Int;
      ___________0030_1 { ExternalAccessible := 'False'; ExternalVisible := 'False'; ExternalWritable := 'False'} : Int;   // ▀▀▀▀ INSTRUMENT TIMER DEFAULT VALUES
      TIME_OPENING_MAX { ExternalWritable := 'False'; S7_SetPoint := 'True'} : Real;   // TIMER — Initial value of opening operation timer [seconds], counts down from this value
      TIME_CLOSING_MAX { ExternalWritable := 'False'; S7_SetPoint := 'True'} : Real;   // TIMER — Initial value of closing operation timer [seconds], counts down from this value
      TIME_FBK_OPEN_SIM { ExternalWritable := 'False'; S7_SetPoint := 'True'} : Real;   // TIMER — Percentage of opening timer to expired before simulating open feedback [percentage]
      TIME_FBK_CLOSED_SIM { ExternalWritable := 'False'; S7_SetPoint := 'True'} : Real;   // TIMER — Percentage of closing timer to expired before simulating closed feedback [percentage]
   END_STRUCT;
   // revInfo.REV_BLOCK := 'UT11001';
   // revInfo.REV_NUMBER := '000.102';
   // revInfo.REV_DATE := '2021-07-21';
   // revInfo.REV_AUTHOR := 'M. Gledhill';
END_TYPE

TYPE "UT11011_St_DevValve3Way"
TITLE = Static UDT [DEVICE DRIVER] — Three-way Valve
// PRACTICAL SERIES AUTOMATION LIBRARY (PAL)   —   COPYRIGHT 2020 – M. GLEDHILL (MIT LICENCE)
//                   ———— ◆ ————
// FULL ONLINE DOCUMENTATION IS AVAILABLE AT: https://practicalseries.com/2001-pal/index.html
// stored: IsFailsafeCompliant false
   STRUCT
      revInfo { ExternalWritable := 'False'} : "UT01000_St_SysRevision";   // Revision information
      ___________0010_0 { ExternalAccessible := 'False'; ExternalVisible := 'False'; ExternalWritable := 'False'} : Int;
      ___________0010_1 { ExternalAccessible := 'False'; ExternalVisible := 'False'; ExternalWritable := 'False'} : Int;   // ▀▀▀▀ INSTRUMENT CONFIGURATION
      CONFIG_FBK_ENG_EN : Bool;   // CONFIG — Energised feedback is enabled (1 = ENG feedback present, 0 = no ENG feedback)
      CONFIG_FBK_DENG_EN : Bool;   // CONFIG — Deenergised feedback is enabled (1 = DENG feedback present, 0 = no DENG feedback)
      CONFIG_ESTOP_DIS : Bool;   // CONFIG — E_STOP signal disabled (1 = E_STOP not used, 0 = E_STOP in use)
      CONFIG_TRIP_DIS : Bool;   // CONFIG — TRIP signal disabled (1 = TRIP not used, 0 = TRIP in use)
      CONFIG_ILOCK_DIS : Bool;   // CONFIG — INTERLOCK signal disabled (1 = INTERLOCK not used, 0 = INTERLOCK in use)
      CONFIG_PERM_DIS : Bool;   // CONFIG — PERMISSIVE signal disabled (1 = PERMISSIVE not used, 0 = PERMISSIVE in use)
      CONFIG_TRIP_ENG_DENG : Bool;   // CONFIG — TRIP state (1 = energised if tripped, 0 = deenergised if tripped)
      CONFIG_ILOCK_ENG_DENG : Bool;   // CONFIG — INTERLOCK state (1 = energised if interlocked, 0 = deenergised if interlocked)
      CONFIG_PERM_ENG_DENG : Bool;   // CONFIG — PERMISSIVE permitted state (1 = permitted energised, 0 = permitted deenergised)
      CONFIG_FP_DIS { ExternalWritable := 'False'; S7_SetPoint := 'True'} : Bool;   // CONFIG — Faceplate is disabled (1 = no Faceplate, 0 = normal)
      CONFIG_MAN_DIS : Bool;   // CONFIG — Manual mode is disabled (1 = no manual mode – auto only, 0 = normal)
      CONFIG_BYPASS_DIS : Bool;   // CONFIG — Bypass mode is disabled (1 = no Bypass, 0 = normal)
      CONFIG_SIM_DIS { ExternalWritable := 'False'; S7_SetPoint := 'True'} : Bool;   // CONFIG — Simulation mode is disabled (1 = no Simulation, 0 = normal)
      CONFIG_RL_EN { ExternalWritable := 'False'; S7_SetPoint := 'True'} : Bool;   // CONFIG — Remote/local mode enabled (1 = remote/local permitted, 0 = remote/local N/A)
      ___________0020_0 { ExternalAccessible := 'False'; ExternalVisible := 'False'; ExternalWritable := 'False'} : Int;
      ___________0020_1 { ExternalAccessible := 'False'; ExternalVisible := 'False'; ExternalWritable := 'False'} : Int;   // ▀▀▀▀ INSTRUMENT INFORMATION (TAG & UNITS)
      INFO_TAG { ExternalWritable := 'False'; S7_SetPoint := 'True'} : String[20];   // INFORMATION — Instrument ID tag
      ___________0030_0 { ExternalAccessible := 'False'; ExternalVisible := 'False'; ExternalWritable := 'False'} : Int;
      ___________0030_1 { ExternalAccessible := 'False'; ExternalVisible := 'False'; ExternalWritable := 'False'} : Int;   // ▀▀▀▀ INSTRUMENT TIMER DEFAULT VALUES
      TIME_ENG_MAX { ExternalWritable := 'False'; S7_SetPoint := 'True'} : Real := 5.0;   // TIMER — Initial value of energising operation timer [seconds], counts down from this value
      TIME_DENG_MAX { ExternalWritable := 'False'; S7_SetPoint := 'True'} : Real := 5.0;   // TIMER — Initial value of deenergising operation timer [seconds], counts down from this value
      TIME_DER_ENG { ExternalWritable := 'False'; S7_SetPoint := 'True'} : Real := 95.0;   // TIMER — Percentage of energising timer to expired before derived ENG feedback [percentage]
      TIME_DER_DENG { ExternalWritable := 'False'; S7_SetPoint := 'True'} : Real := 95.0;   // TIMER — Percentage of deenergising timer to expired before derived DENG feedback [percentage]
   END_STRUCT;
   // revInfo.REV_BLOCK := 'UT11011';
   // revInfo.REV_NUMBER := '000.801';
   // revInfo.REV_DATE := '2022.06.07';
   // revInfo.REV_AUTHOR := 'M. Gledhill';
END_TYPE

TYPE "UT11101_St_DevValveBi"
TITLE = Static UDT [DEVICE DRIVER] — Bistable Valve
// PRACTICAL SERIES AUTOMATION LIBRARY (PAL)   —   COPYRIGHT 2020 – M. GLEDHILL (MIT LICENCE)
//                   ———— ◆ ————
// FULL ONLINE DOCUMENTATION IS AVAILABLE AT: https://practicalseries.com/2001-pal/index.html
// stored: IsFailsafeCompliant false
   STRUCT
      revInfo { ExternalWritable := 'False'} : "UT01000_St_SysRevision";   // Revision information
      ___________0010_0 { ExternalAccessible := 'False'; ExternalVisible := 'False'; ExternalWritable := 'False'} : Int;
      ___________0010_1 { ExternalAccessible := 'False'; ExternalVisible := 'False'; ExternalWritable := 'False'} : Int;   // ▀▀▀▀ INSTRUMENT CONFIGURATION
      CONFIG_MAINT_OP : Bool;   // CONFIG — Maintains or deenergises the outputs (1 = maintain OP, 0 = deenergise OP)
      CONFIG_FBK_OPEN_EN : Bool;   // CONFIG — Open feedback is enabled (1 = open feedback present, 0 = no open feedback)
      CONFIG_FBK_CLOSED_EN : Bool;   // CONFIG — Closed feedback is enabled (1 = closed feedback present, 0 = no closed feedback)
      CONFIG_ESTOP_DIS : Bool;   // CONFIG — E_STOP signal disabled (1 = E_STOP not used, 0 = E_STOP in use)
      CONFIG_TRIP_DIS : Bool;   // CONFIG — TRIP signal disabled (1 = TRIP not used, 0 = TRIP in use)
      CONFIG_ILOCK_DIS : Bool;   // CONFIG — INTERLOCK signal disabled (1 = INTERLOCK not used, 0 = INTERLOCK in use)
      CONFIG_PERM_DIS : Bool;   // CONFIG — PERMISSIVE signal disabled (1 = PERMISSIVE not used, 0 = PERMISSIVE in use)
      CONFIG_TRIP_OP_CL : Bool;   // CONFIG — TRIP state (1 = open if tripped, 0 = close if tripped)
      CONFIG_ILOCK_OP_CL : Bool;   // CONFIG — INTERLOCK state (1 = open if interlocked, 0 = close if interlocked)
      CONFIG_PERM_OP_CL : Bool;   // CONFIG — PERMISSIVE permitted state (1 = permitted state open, 0 = permitted state closed)
      CONFIG_FP_DIS { ExternalWritable := 'False'; S7_SetPoint := 'True'} : Bool;   // CONFIG — Faceplate is disabled (1 = no Faceplate, 0 = normal)
      CONFIG_MAN_DIS : Bool;   // CONFIG — Manual mode is disabled (1 = no manual mode – auto only, 0 = normal)
      CONFIG_BYPASS_DIS : Bool;   // CONFIG — Bypass mode is disabled (1 = no Bypass, 0 = normal)
      CONFIG_SIM_DIS { ExternalWritable := 'False'; S7_SetPoint := 'True'} : Bool;   // CONFIG — Simulation mode is disabled (1 = no Simulation, 0 = normal)
      CONFIG_RL_EN { ExternalWritable := 'False'; S7_SetPoint := 'True'} : Bool;   // CONFIG — Remote/local mode enabled (1 = remote/local permitted, 0 = remote/local N/A)
      ___________0020_0 { ExternalAccessible := 'False'; ExternalVisible := 'False'; ExternalWritable := 'False'} : Int;
      ___________0020_1 { ExternalAccessible := 'False'; ExternalVisible := 'False'; ExternalWritable := 'False'} : Int;   // ▀▀▀▀ INSTRUMENT INFORMATION (TAG & UNITS)
      INFO_TAG { ExternalWritable := 'False'; S7_SetPoint := 'True'} : String[20];   // INFORMATION — Instrument ID tag
      ___________0030_0 { ExternalAccessible := 'False'; ExternalVisible := 'False'; ExternalWritable := 'False'} : Int;
      ___________0030_1 { ExternalAccessible := 'False'; ExternalVisible := 'False'; ExternalWritable := 'False'} : Int;   // ▀▀▀▀ INSTRUMENT TIMER DEFAULT VALUES
      TIME_OPENING_MAX { ExternalWritable := 'False'; S7_SetPoint := 'True'} : Real := 5.0;   // TIMER — Initial value of opening operation timer [seconds], counts down from this value
      TIME_CLOSING_MAX { ExternalWritable := 'False'; S7_SetPoint := 'True'} : Real := 5.0;   // TIMER — Initial value of closing operation timer [seconds], counts down from this value
      TIME_OPENING_RUNON { ExternalWritable := 'False'; S7_SetPoint := 'True'} : Real := 2.0;   // TIMER — Initial value of opening run-on timer [seconds], counts down from this value
      TIME_CLOSING_RUNON { ExternalWritable := 'False'; S7_SetPoint := 'True'} : Real := 2.0;   // TIMER — Initial value of closing run-on timer [seconds], counts down from this value
      TIME_DER_OPEN { ExternalWritable := 'False'; S7_SetPoint := 'True'} : Real := 95.0;   // TIMER — Percentage of opening timer to expired before derived open feedback [percentage]
      TIME_DER_CLOSED { ExternalWritable := 'False'; S7_SetPoint := 'True'} : Real := 95.0;   // TIMER — Percentage of closing timer to expired before derived closed feedback [percentage]
      TIME_RECOVERY { ExternalWritable := 'False'; S7_SetPoint := 'True'} : Real := 5.0;   // TIMER — Initial value of the recovery timer [seconds], counts down from this value
   END_STRUCT;
   // revInfo.REV_BLOCK := 'UT11101';
   // revInfo.REV_NUMBER := '000.801';
   // revInfo.REV_DATE := '2023.02.01';
   // revInfo.REV_AUTHOR := 'M. Gledhill';
END_TYPE

TYPE "UT31001_Dy_DevValveIsol"
TITLE = Dynamic UDT [Instrumentation] — Analog Instrument Read, Scale and Monitor
// Analogue Instrument Read and Scale
// stored: IsFailsafeCompliant false
   STRUCT
      revInfo : "UT01000_St_SysRevision";   // Revision information
      ___________0010_0 { ExternalAccessible := 'False'; ExternalVisible := 'False'; ExternalWritable := 'False'} : Int;
      ___________0010_1 { ExternalAccessible := 'False'; ExternalVisible := 'False'; ExternalWritable := 'False'} : Int;   // ▀▀▀▀ STATUS (FOR BLOCK ICON AND SYMBOL)
      status_Closed : Bool;   // STATUS — Valve is confirmed closed (1 = valve is closed, 0 = valve is not closed)
      status_Open : Bool;   // STATUS — Valve is confirmed open (1 = valve is open, 0 = valve is not open)
      status_Closing : Bool;   // STATUS — Valve is closing (1 = valve is closing, 0 = valve is not closing)
      status_Opening : Bool;   // STATUS — Valve is opening (1 = valve is opening, 0 = valve is not opening)
      status_Operating : Bool;   // STATUS — Valve is changing state (1 = valve is opening or closing, 0 = valve is not moving)
      status_Fault : Bool;   // STATUS — Valve is in fault (1 = fault present, 0 = healthy)
      status_Energised : Bool;   // STATUS — Valve output is on (1 = valve energised, 0 = valve deenergised)
      status_Aut : Bool;   // STATUS — Automatic mode active (1 = in automatic mode, 0 = not in automatic mode)
      status_Man : Bool;   // STATUS — Manual mode active (1 = in manual mode, 0 = not in manual mode)
      status_EStop : Bool;   // STATUS — E_STOP safety signal is active (1 = E_STOP active, 0 = E_STOP not active)
      status_Trip : Bool;   // STATUS — TRIP signal is active (1 = TRIP active, 0 = TRIP not active)
      status_Ilock : Bool;   // STATUS — INTERLOCK signal is active (1 = INTERLOCK active, 0 = INTERLOCK not active)
      status_Perm : Bool;   // STATUS — PERMISSIVE signal is active (1 = PERMISSIVE active, 0 = PERMISSIVE not active)
      status_BypassOn : Bool;   // STATUS — Valve is in bypass mode (1 = bypass mode on, 0 = normal)
      status_SimOn : Bool;   // STATUS — Valve is in simulation mode (1 = simulation mode on, 0 = normal)
      status_RemoteOn : Bool;   // STATUS — Valve is in remote mode (1 = remote mode, 0 = remote mode off)
      status_LocalOn : Bool;   // STATUS — Valve is in local mode (1 = local mode, 0 = local mode off)
      status_RLOff : Bool;   // STATUS — Remote/local mode disabled (1 = ALL mode on, 0 = RL mode selected)
      ___________0020_0 { ExternalAccessible := 'False'; ExternalVisible := 'False'; ExternalWritable := 'False'} : Int;
      ___________0020_1 { ExternalAccessible := 'False'; ExternalVisible := 'False'; ExternalWritable := 'False'} : Int;   // ▀▀▀▀ MESSAGES (ALARMS, WARNINGS, FAULTS AND EVENTS)
      msg_FailToOpen : Bool;   // MESSAGE — Alarm – “Fail to open” is active (1 = alarm active, 0 = alarm not active)
      msg_FailToClose : Bool;   // MESSAGE — Alarm – “Fail to close” is active (1 = alarm active, 0 = alarm not active)
      msg_FailWhileOpen : Bool;   // MESSAGE — Alarm – “Fail while open” is active (1 = alarm active, 0 = alarm not active)
      msg_FailWhileClosed : Bool;   // MESSAGE — Alarm – “Fail while closed” is active (1 = alarm active, 0 = alarm not active)
      msg_Flt_External : Bool;   // MESSAGE — Alarm – “External fault” is active (1 = alarm active, 0 = alarm not active)
      ___________0030_0 { ExternalAccessible := 'False'; ExternalVisible := 'False'; ExternalWritable := 'False'} : Int;
      ___________0030_1 { ExternalAccessible := 'False'; ExternalVisible := 'False'; ExternalWritable := 'False'} : Int;   // ▀▀▀▀ OPERATING MODE SELECTION (FROM FACEPLATE OR PANEL)
      mode_AutMan : Bool;   // MODE — Automatic or manual mode selection (1 = automatic mode, 0 = manual mode)
      mode_BypassOn : Bool;   // MODE — Bypass mode (1 = bypass mode active, 0 = normal)
      mode_SimOn : Bool;   // MODE — Simulation mode (1 = simulation mode active, 0 = normal)
      mode_SimValue : Int;   // MODE — Simulation value (0 no limits, 1 always open, 2 always closed, 3 follow demand)
      mode_RemoteOn : Bool;   // MODE — Local HMI control enabled (1 = control active, 0 = control disabled or N/A)
      mode_LocalOn : Bool;   // MODE — Remote SCADA control enabled (1 = control active, 0 = control disabled or N/A)
      mode_Reset : Bool;   // MODE — Fault reset (1 = Reset any faults – 1 cycle only, 0 = does nothing)
      ___________0040_0 { ExternalAccessible := 'False'; ExternalVisible := 'False'; ExternalWritable := 'False'} : Int;
      ___________0040_1 { ExternalAccessible := 'False'; ExternalVisible := 'False'; ExternalWritable := 'False'} : Int;   // ▀▀▀▀ CONTROL SIGNALS (TO OPERATE THE DEVICE)
      ctrl_Aut_OpenClose : Bool;   // CONTROL — Auto mode open or close valve (1 = open valve in auto, 0 = close valve in auto)
      ctrl_Man_OpenClose : Bool;   // CONTROL — Manual mode open or close valve (1 = open valve in man, 0 = close valve in man)
      ___________0050_0 { ExternalAccessible := 'False'; ExternalVisible := 'False'; ExternalWritable := 'False'} : Int;
      ___________0050_1 { ExternalAccessible := 'False'; ExternalVisible := 'False'; ExternalWritable := 'False'} : Int;   // ▀▀▀▀ BATCH AND BOOKING DATA
      batch_ID : Int;   // BATCH — Booking ID (optional for batch operations)
      ___________0060_0 { ExternalAccessible := 'False'; ExternalVisible := 'False'; ExternalWritable := 'False'} : Int;
      ___________0060_1 { ExternalAccessible := 'False'; ExternalVisible := 'False'; ExternalWritable := 'False'} : Int;   // ▀▀▀▀ LIVE DATA (SCALED READING & TIMER VALUES)
      actual_Operating_Timer : Real;   // ACTUAL — Timer value — operating opening/closing timer actual value [seconds]
      ___________0090_0 { ExternalAccessible := 'False'; ExternalVisible := 'False'; ExternalWritable := 'False'} : Int;
      ___________0090_1 { ExternalAccessible := 'False'; ExternalVisible := 'False'; ExternalWritable := 'False'} : Int;   // ▀▀▀▀ BLOCK INTERNAL WORKING AND STORAGE AREA
      "$derived_fbk_open" : Bool;   // INTERNAL — Derived feedback open signal (if CONFIG_FBK_OPEN_EN = 0)
      "$derived_fbk_closed" : Bool;   // INTERNAL — Derived feedback closed signal (if CONFIG_FBK_CLOSED_EN = 0)
      "$sim_fbk_open" : Bool;   // INTERNAL — Simulated feedback open signal (if mode_SimOn = 1)
      "$sim_fbk_closed" : Bool;   // INTERNAL — Simulated feedback closed signal (if mode_SimOn = 1)
      "$ctrl_OpenClose" : Bool;   // INTERNAL — actual open or close control signal passed to the valve (1 = open, 0 = close)
      "$pret_Open" : Bool;   // INTERNAL — Edge retention (+ve) rising edge of ctrl_OpenClose (change of state to open)
      "$nret_Close" : Bool;   // INTERNAL — Edge retention (-ve) falling edge of ctrl_OpenClose (change of state to close)
   END_STRUCT;
   // revInfo.REV_BLOCK := 'UT31001';
   // revInfo.REV_NUMBER := '000.102';
   // revInfo.REV_DATE := '2021-07-21';
   // revInfo.REV_AUTHOR := 'M. Gledhill';
END_TYPE

TYPE "UT31011_Dy_DevValve3Way"
TITLE = Dynamic UDT [DEVICE DRIVER] — Three-way Valve
// PRACTICAL SERIES AUTOMATION LIBRARY (PAL)   —   COPYRIGHT 2020 – M. GLEDHILL (MIT LICENCE)
//                   ———— ◆ ————
// FULL ONLINE DOCUMENTATION IS AVAILABLE AT: https://practicalseries.com/2001-pal/index.html
// stored: IsFailsafeCompliant false
   STRUCT
      revInfo : "UT01000_St_SysRevision";   // Revision information
      ___________0010_0 { ExternalAccessible := 'False'; ExternalVisible := 'False'; ExternalWritable := 'False'} : Int;
      ___________0010_1 { ExternalAccessible := 'False'; ExternalVisible := 'False'; ExternalWritable := 'False'} : Int;   // ▀▀▀▀ STATUS (FOR BLOCK ICON AND SYMBOL)
      status_Deenergised : Bool;   // STATUS — Valve is confirmed deenergised (1 = valve is in deenergised state)
      status_Energised : Bool;   // STATUS — Valve is confirmed energised (1 = valve is in energised state)
      status_Deenergising : Bool;   // STATUS — Valve is deenergising (1 = valve is deenergising, 0 = valve is not deenergising)
      status_Energising : Bool;   // STATUS — Valve is energising (1 = valve is energising, 0 = valve is not energising)
      status_Operating : Bool;   // STATUS — Valve is changing state (1 = valve is energising or deenergising, 0 = valve is not moving)
      status_Fault { ExternalWritable := 'False'} : Bool;   // STATUS — Valve is in fault (1 = fault present, 0 = healthy)
      status_OperateOn : Bool;   // STATUS — Valve output is on (1 = valve energised, 0 = valve deenergised)
      status_Aut : Bool;   // STATUS — Automatic mode active (1 = in automatic mode, 0 = not in automatic mode)
      status_Man : Bool;   // STATUS — Manual mode active (1 = in manual mode, 0 = not in manual mode)
      status_EStop : Bool;   // STATUS — E_STOP safety signal is active (1 = E_STOP active, 0 = E_STOP not active)
      status_Trip : Bool;   // STATUS — TRIP signal is active (1 = TRIP active, 0 = TRIP not active)
      status_Ilock : Bool;   // STATUS — INTERLOCK signal is active (1 = INTERLOCK active, 0 = INTERLOCK not active)
      status_Perm : Bool;   // STATUS — PERMISSIVE signal is active (1 = PERMISSIVE active, 0 = PERMISSIVE not active)
      status_BypassOn : Bool;   // STATUS — Valve is in bypass mode (1 = bypass mode on, 0 = normal)
      status_SimOn : Bool;   // STATUS — Valve is in simulation mode (1 = simulation mode on, 0 = normal)
      status_RemoteOn : Bool;   // STATUS — Valve is in remote mode (1 = remote mode, 0 = remote mode off)
      status_LocalOn : Bool;   // STATUS — Valve is in local mode (1 = local mode, 0 = local mode off)
      status_RLOff : Bool;   // STATUS — Remote/local mode disabled (1 = ALL mode on, 0 = RL mode selected)
      ___________0020_0 { ExternalAccessible := 'False'; ExternalVisible := 'False'; ExternalWritable := 'False'} : Int;
      ___________0020_1 { ExternalAccessible := 'False'; ExternalVisible := 'False'; ExternalWritable := 'False'} : Int;   // ▀▀▀▀ MESSAGES (ALARMS, WARNINGS, FAULTS AND EVENTS)
      msg_FailToEnergise : Bool;   // MESSAGE — Alarm – “Fail to energise” is active (1 = alarm active, 0 = alarm not active)
      msg_FailToDeenergise : Bool;   // MESSAGE — Alarm – “Fail to deenergise” is active (1 = alarm active, 0 = alarm not active)
      msg_FailWhileEnergised : Bool;   // MESSAGE — Alarm – “Fail while energised” is active (1 = alarm active, 0 = alarm not active)
      msg_FailWhileDeenergised : Bool;   // MESSAGE — Alarm – “Fail while deenergised” is active (1 = alarm active, 0 = alarm not active)
      msg_Flt_External : Bool;   // MESSAGE — Alarm – “External fault” is active (1 = alarm active, 0 = alarm not active)
      ___________0030_0 { ExternalAccessible := 'False'; ExternalVisible := 'False'; ExternalWritable := 'False'} : Int;
      ___________0030_1 { ExternalAccessible := 'False'; ExternalVisible := 'False'; ExternalWritable := 'False'} : Int;   // ▀▀▀▀ OPERATING MODE SELECTION (FROM FACEPLATE OR PANEL)
      mode_AutMan : Bool := true;   // MODE — Automatic or manual mode selection (1 = automatic mode, 0 = manual mode)
      mode_BypassOn : Bool;   // MODE — Bypass mode (1 = bypass mode active, 0 = normal)
      mode_SimOn : Bool;   // MODE — Simulation mode (1 = simulation mode active, 0 = normal)
      mode_SimValue : Int;   // MODE — Simulation value (0 no limits, 1 always open, 2 always closed, 3 follow demand)
      mode_RemoteOn : Bool;   // MODE — Local HMI control enabled (1 = control active, 0 = control disabled or N/A)
      mode_LocalOn : Bool;   // MODE — Remote SCADA control enabled (1 = control active, 0 = control disabled or N/A)
      mode_Reset : Bool;   // MODE — Fault reset (1 = Reset any faults – 1 cycle only, 0 = does nothing)
      ___________0040_0 { ExternalAccessible := 'False'; ExternalVisible := 'False'; ExternalWritable := 'False'} : Int;
      ___________0040_1 { ExternalAccessible := 'False'; ExternalVisible := 'False'; ExternalWritable := 'False'} : Int;   // ▀▀▀▀ CONTROL SIGNALS (TO OPERATE THE DEVICE)
      ctrl_Aut_EngDeng : Bool;   // CONTROL — Auto mode energise or deenergise valve (1 = energise in auto, 0 = deenergise in auto)
      ctrl_Man_EngDeng : Bool;   // CONTROL — Manual mode energise or deenergise valve (1 = energise in man, 0 = deenergise in man)
      ___________0050_0 { ExternalAccessible := 'False'; ExternalVisible := 'False'; ExternalWritable := 'False'} : Int;
      ___________0050_1 { ExternalAccessible := 'False'; ExternalVisible := 'False'; ExternalWritable := 'False'} : Int;   // ▀▀▀▀ BATCH AND BOOKING DATA
      batch_ID : UInt;   // BATCH — Booking ID (optional for batch operations)
      ___________0060_0 { ExternalAccessible := 'False'; ExternalVisible := 'False'; ExternalWritable := 'False'} : Int;
      ___________0060_1 { ExternalAccessible := 'False'; ExternalVisible := 'False'; ExternalWritable := 'False'} : Int;   // ▀▀▀▀ LIVE DATA (SCALED READING & TIMER VALUES)
      actual_Operating_Timer : Real;   // ACTUAL — Timer value — operating energising/deenergising timer actual value [seconds]
      actual_Last_Op_Time : Real;   // ACTUAL — Timer value — last operation time before feedback [seconds]
      ___________0090_0 { ExternalAccessible := 'False'; ExternalVisible := 'False'; ExternalWritable := 'False'} : Int;
      ___________0090_1 { ExternalAccessible := 'False'; ExternalVisible := 'False'; ExternalWritable := 'False'} : Int;   // ▀▀▀▀ BLOCK INTERNAL WORKING AND STORAGE AREA
      "$derived_fbk_eng" : Bool;   // INTERNAL — Derived feedback ENG signal (if CONFIG_FBK_ENG_EN = 0)
      "$derived_fbk_deng" : Bool;   // INTERNAL — Derived feedback DENG signal (if CONFIG_FBK_DENG_EN = 0)
      "$sim_fbk_eng" : Bool;   // INTERNAL — Simulated feedback ENG signal (if mode_SimOn = 1)
      "$sim_fbk_deng" : Bool;   // INTERNAL — Simulated feedback DENG signal (if mode_SimOn = 1)
      "$ctrl_EngDeng" : Bool;   // INTERNAL — actual energise or deenergise control signal passed to the valve (1 = eng, 0 = deng)
      "$pret_eng" : Bool;   // INTERNAL — Edge retention (+ve) rising edge of ctrl_OpenClose (change of state to energising)
      "$nret_deng" : Bool;   // INTERNAL — Edge retention (-ve) falling edge of ctrl_OpenClose (change of state to deenergising)
   END_STRUCT;
   // revInfo.REV_BLOCK := 'UT31011';
   // revInfo.REV_NUMBER := '000.801';
   // revInfo.REV_DATE := '2022.06.07';
   // revInfo.REV_AUTHOR := 'M. Gledhill';
END_TYPE

TYPE "UT31101_Dy_DevValveBi"
TITLE = Dynamic UDT [DEVICE DRIVER] — Bistable Valve
// PRACTICAL SERIES AUTOMATION LIBRARY (PAL)   —   COPYRIGHT 2020 – M. GLEDHILL (MIT LICENCE)
//                   ———— ◆ ————
// FULL ONLINE DOCUMENTATION IS AVAILABLE AT: https://practicalseries.com/2001-pal/index.html
// stored: IsFailsafeCompliant false
   STRUCT
      revInfo : "UT01000_St_SysRevision";   // Revision information
      ___________0010_0 { ExternalAccessible := 'False'; ExternalVisible := 'False'; ExternalWritable := 'False'} : Int;
      ___________0010_1 { ExternalAccessible := 'False'; ExternalVisible := 'False'; ExternalWritable := 'False'} : Int;   // ▀▀▀▀ STATUS (FOR BLOCK ICON AND SYMBOL)
      status_Closed : Bool;   // STATUS — Valve is confirmed closed (1 = valve is closed, 0 = valve is not closed)
      status_Open : Bool;   // STATUS — Valve is confirmed open (1 = valve is open, 0 = valve is not open)
      status_Closing : Bool;   // STATUS — Valve is closing (1 = valve is closing, 0 = valve is not closing)
      status_Opening : Bool;   // STATUS — Valve is opening (1 = valve is opening, 0 = valve is not opening)
      status_Operating : Bool;   // STATUS — Valve is changing state (1 = valve is opening or closing, 0 = valve is not moving)
      status_Fault { ExternalWritable := 'False'} : Bool;   // STATUS — Valve is in fault (1 = fault present, 0 = healthy)
      status_Energised : Bool;   // STATUS — Valve output is on (1 = valve energised, 0 = valve deenergised)
      status_Aut : Bool;   // STATUS — Automatic mode active (1 = in automatic mode, 0 = not in automatic mode)
      status_Man : Bool;   // STATUS — Manual mode active (1 = in manual mode, 0 = not in manual mode)
      status_EStop : Bool;   // STATUS — E_STOP safety signal is active (1 = E_STOP active, 0 = E_STOP not active)
      status_Trip : Bool;   // STATUS — TRIP signal is active (1 = TRIP active, 0 = TRIP not active)
      status_Ilock : Bool;   // STATUS — INTERLOCK signal is active (1 = INTERLOCK active, 0 = INTERLOCK not active)
      status_Perm : Bool;   // STATUS — PERMISSIVE signal is active (1 = PERMISSIVE active, 0 = PERMISSIVE not active)
      status_BypassOn : Bool;   // STATUS — Valve is in bypass mode (1 = bypass mode on, 0 = normal)
      status_SimOn : Bool;   // STATUS — Valve is in simulation mode (1 = simulation mode on, 0 = normal)
      status_RemoteOn : Bool;   // STATUS — Valve is in remote mode (1 = remote mode, 0 = remote mode off)
      status_LocalOn : Bool;   // STATUS — Valve is in local mode (1 = local mode, 0 = local mode off)
      status_RLOff : Bool;   // STATUS — Remote/local mode disabled (1 = ALL mode on, 0 = RL mode selected)
      ___________0020_0 { ExternalAccessible := 'False'; ExternalVisible := 'False'; ExternalWritable := 'False'} : Int;
      ___________0020_1 { ExternalAccessible := 'False'; ExternalVisible := 'False'; ExternalWritable := 'False'} : Int;   // ▀▀▀▀ MESSAGES (ALARMS, WARNINGS, FAULTS AND EVENTS)
      msg_FailToOpen : Bool;   // MESSAGE — Alarm – “Fail to open” is active (1 = alarm active, 0 = alarm not active)
      msg_FailToClose : Bool;   // MESSAGE — Alarm – “Fail to close” is active (1 = alarm active, 0 = alarm not active)
      msg_FailWhileOpen : Bool;   // MESSAGE — Alarm – “Fail while open” is active (1 = alarm active, 0 = alarm not active)
      msg_FailWhileClosed : Bool;   // MESSAGE — Alarm – “Fail while closed” is active (1 = alarm active, 0 = alarm not active)
      msg_Flt_External : Bool;   // MESSAGE — Alarm – “External fault” is active (1 = alarm active, 0 = alarm not active)
      ___________0030_0 { ExternalAccessible := 'False'; ExternalVisible := 'False'; ExternalWritable := 'False'} : Int;
      ___________0030_1 { ExternalAccessible := 'False'; ExternalVisible := 'False'; ExternalWritable := 'False'} : Int;   // ▀▀▀▀ OPERATING MODE SELECTION (FROM FACEPLATE OR PANEL)
      mode_AutMan : Bool := true;   // MODE — Automatic or manual mode selection (1 = automatic mode, 0 = manual mode)
      mode_BypassOn : Bool;   // MODE — Bypass mode (1 = bypass mode active, 0 = normal)
      mode_SimOn : Bool;   // MODE — Simulation mode (1 = simulation mode active, 0 = normal)
      mode_SimValue : Int;   // MODE — Simulation value (0 no limits, 1 always open, 2 always closed, 3 follow demand)
      mode_RemoteOn : Bool;   // MODE — Local HMI control enabled (1 = control active, 0 = control disabled or N/A)
      mode_LocalOn : Bool;   // MODE — Remote SCADA control enabled (1 = control active, 0 = control disabled or N/A)
      mode_Reset : Bool;   // MODE — Fault reset (1 = Reset any faults – 1 cycle only, 0 = does nothing)
      ___________0040_0 { ExternalAccessible := 'False'; ExternalVisible := 'False'; ExternalWritable := 'False'} : Int;
      ___________0040_1 { ExternalAccessible := 'False'; ExternalVisible := 'False'; ExternalWritable := 'False'} : Int;   // ▀▀▀▀ CONTROL SIGNALS (TO OPERATE THE DEVICE)
      ctrl_Aut_OpenClose : Bool;   // CONTROL — Auto mode open or close valve (1 = open valve in auto, 0 = close valve in auto)
      ctrl_Man_OpenClose : Bool;   // CONTROL — Manual mode open or close valve (1 = open valve in man, 0 = close valve in man)
      ___________0050_0 { ExternalAccessible := 'False'; ExternalVisible := 'False'; ExternalWritable := 'False'} : Int;
      ___________0050_1 { ExternalAccessible := 'False'; ExternalVisible := 'False'; ExternalWritable := 'False'} : Int;   // ▀▀▀▀ BATCH AND BOOKING DATA
      batch_ID : UInt;   // BATCH — Booking ID (optional for batch operations)
      ___________0060_0 { ExternalAccessible := 'False'; ExternalVisible := 'False'; ExternalWritable := 'False'} : Int;
      ___________0060_1 { ExternalAccessible := 'False'; ExternalVisible := 'False'; ExternalWritable := 'False'} : Int;   // ▀▀▀▀ LIVE DATA (SCALED READING & TIMER VALUES)
      actual_Operating_Timer : Real;   // ACTUAL — Timer value — operating opening/closing timer actual value [seconds]
      actual_Last_Op_Time : Real;   // ACTUAL — Timer value — last operation time before feedback [seconds]
      ___________0090_0 { ExternalAccessible := 'False'; ExternalVisible := 'False'; ExternalWritable := 'False'} : Int;
      ___________0090_1 { ExternalAccessible := 'False'; ExternalVisible := 'False'; ExternalWritable := 'False'} : Int;   // ▀▀▀▀ BLOCK INTERNAL WORKING AND STORAGE AREA
      "$derived_fbk_open" : Bool;   // INTERNAL — Derived feedback open signal (if CONFIG_FBK_OPEN_EN = 0)
      "$derived_fbk_closed" : Bool;   // INTERNAL — Derived feedback closed signal (if CONFIG_FBK_CLOSED_EN = 0)
      "$sim_fbk_open" : Bool;   // INTERNAL — Simulated feedback open signal (if mode_SimOn = 1)
      "$sim_fbk_closed" : Bool;   // INTERNAL — Simulated feedback closed signal (if mode_SimOn = 1)
      "$ctrl_OpenClose" : Bool;   // INTERNAL — actual open or close control signal passed to the valve (1 = open, 0 = close)
      "$pret_Open" : Bool;   // INTERNAL — Edge retention (+ve) rising edge of ctrl_OpenClose (change of state to open)
      "$nret_Close" : Bool;   // INTERNAL — Edge retention (-ve) falling edge of ctrl_OpenClose (change of state to close)
   END_STRUCT;
   // revInfo.REV_BLOCK := 'UT31001';
   // revInfo.REV_NUMBER := '000.101';
   // revInfo.REV_DATE := '2022.08.15';
   // revInfo.REV_AUTHOR := 'M. Gledhill';
END_TYPE

TYPE "UT39511_Dy_DebugInst1Order"
TITLE = Dynamic UDT [DEBUG] — First Order Response Simulation
// PRACTICAL SERIES AUTOMATION LIBRARY (PAL)   —   COPYRIGHT 2020 – M. GLEDHILL (MIT LICENCE)
//                   ———— ◆ ————
// FULL ONLINE DOCUMENTATION IS AVAILABLE AT: https://practicalseries.com/2001-pal/index.html
// stored: IsFailsafeCompliant false
   STRUCT
      revInfo { ExternalWritable := 'False'} : "UT01000_St_SysRevision";   // ▀▀▀▀ UDT CURRENT REVISION
      ___________0010_0 { ExternalAccessible := 'False'; ExternalVisible := 'False'; ExternalWritable := 'False'} : Int;
      ___________0010_1 { ExternalAccessible := 'False'; ExternalVisible := 'False'; ExternalWritable := 'False'} : Int;   // ▀▀▀▀ CALCULATION CONSTANTS
      k_Gain : Real := 1.0;   // CONSTANT — Simulation system gain
      k_TimeConstant : Real := 1.0;   // CONSTANT — Simulation system time constant (s)
      ___________0020_0 { ExternalAccessible := 'False'; ExternalVisible := 'False'; ExternalWritable := 'False'} : Int;
      ___________0020_1 { ExternalAccessible := 'False'; ExternalVisible := 'False'; ExternalWritable := 'False'} : Int;   // ▀▀▀▀ SIMULATION STATUS SIGNALS
      status_Running : Bool;   // STATUS — Simulation is running (1 = running, 0 = stopped)
      status_Stopped : Bool;   // STATUS — Simulation is stopped (not running) (1 = stopped, 0 = running)
      status_SteadyState : Bool;   // STATUS — Steady state (±2%) achieved (1 = In steady state, 0 = not steady state)
      status_Aut : Bool;   // STATUS — Simulation is in automatic mode (1 = automatic, 0 = manual)
      status_Man : Bool;   // STATUS — Simulation is in manual mode (1 = manual, 0 = automatic)
      ___________0030_0 { ExternalAccessible := 'False'; ExternalVisible := 'False'; ExternalWritable := 'False'} : Int;
      ___________0030_1 { ExternalAccessible := 'False'; ExternalVisible := 'False'; ExternalWritable := 'False'} : Int;   // ▀▀▀▀ CALCULATED VALUES
      cal_TimeSteady : Real;   // CALC — Time to reach steady state, zero for unstable response (s)
      ___________0040_0 { ExternalAccessible := 'False'; ExternalVisible := 'False'; ExternalWritable := 'False'} : Int;
      ___________0040_1 { ExternalAccessible := 'False'; ExternalVisible := 'False'; ExternalWritable := 'False'} : Int;   // ▀▀▀▀ OPERATING MODE SELECTION
      mode_AutMan : Bool := true;   // MODE — Automatic/manual mode selection (1 = auto mode, 0 = manual mode)
      mode_ManTime : Real;   // MODE — Manual mode time value (s)
      ___________0050_0 { ExternalAccessible := 'False'; ExternalVisible := 'False'; ExternalWritable := 'False'} : Int;
      ___________0050_1 { ExternalAccessible := 'False'; ExternalVisible := 'False'; ExternalWritable := 'False'} : Int;   // ▀▀▀▀ LIVE TIMING DATA
      actual_Output : Real;   // ACTUAL — SIMULATION OUTPUT VALUE (identical to OUTPUT parameter)
      actual_PrevOutput : Real;   // ACTUAL — Output value from the previous iteration y[n-1]
      actual_StartTime : DTL;   // ACTUAL — CPU time when simulation started
      actual_Time : DTL;   // ACTUAL — CPU time of this (current) iteration of the calculation
      actual_PrevTime : DTL;   // ACTUAL — CPU time of the previous iteration of the calculation
      actual_RunTime : Real;   // ACTUAL — Elapsed time since the simulation started (s)
      actual_DeltaTime : Real;   // ACTUAL — Time period between this and previous iteration (s)
   END_STRUCT;
   // revInfo.REV_BLOCK := 'UT39511';
   // revInfo.REV_NUMBER := '001.000';
   // revInfo.REV_DATE := '2023-03-03';
   // revInfo.REV_AUTHOR := 'M. Gledhill';
END_TYPE

TYPE "UT39512_Dy_DebugInst2Order"
TITLE = Dynamic UDT [Debug] — Second Order Response Simulation
// Second Order Response Simulation
// stored: IsFailsafeCompliant false
   STRUCT
      revInfo { ExternalWritable := 'False'} : "UT01000_St_SysRevision";   // ▀▀▀▀ UDT CURRENT REVISION
      ___________0010_0 { ExternalAccessible := 'False'; ExternalVisible := 'False'; ExternalWritable := 'False'} : Int;
      ___________0010_1 { ExternalAccessible := 'False'; ExternalVisible := 'False'; ExternalWritable := 'False'} : Int;   // ▀▀▀▀ CALCULATION CONSTANTS
      k_Gain : Real;   // CONSTANT — Simulation system gain
      k_NatFreq : Real;   // CONSTANT — Simulation natural frequency (rad/s)
      k_DampFactor : Real;   // CONSTANT — Simulation damping factor
      ___________0020_0 { ExternalAccessible := 'False'; ExternalVisible := 'False'; ExternalWritable := 'False'} : Int;
      ___________0020_1 { ExternalAccessible := 'False'; ExternalVisible := 'False'; ExternalWritable := 'False'} : Int;   // ▀▀▀▀ SIMULATION STATUS SIGNALS
      status_Running : Bool;   // STATUS — Simulation is running (1 = running, 0 = stopped)
      status_Stopped : Bool;   // STATUS — Simulation is stopped (not running) (1 = stopped, 0 = running)
      status_Stable : Bool;   // STATUS — Simulation response type is stable (1 = stable, 0 = unstable)
      status_OverDamp : Bool;   // STATUS — Response is stable/over damped (1 = stable, over damped)
      status_CritDamp : Bool;   // STATUS — Response is stable/critically damped (1 = stable, critically damped)
      status_UnderDamp : Bool;   // STATUS — Response is stable/under damped (1 = stable, under damped)
      status_Undamped : Bool;   // STATUS — Response is stable/undamped (1 = stable, undamped)
      status_USUnder : Bool;   // STATUS — Response is unstable/under damped (1 = unstable, under damped)
      status_USOver : Bool;   // STATUS — Response is unstable/over damped (1 = unstable, over damped)
      status_SteadyState : Bool;   // STATUS — Steady state (±2%) achieved (1 = In steady state, 0 = not steady state)
      status_Osc : Bool;   // STATUS — Oscillatory response (1 = oscillating response, 0 = non-oscillating)
      status_OscFreqRS : Real;   // STATUS — Frequency of oscillation, zero if non oscillatory (rad/s)
      status_OscFreqHz : Real;   // STATUS — Frequency of oscillation, zero if non oscillatory (Hz)
      status_Period : Real;   // STATUS — Period of oscillation, zero if non oscillatory (s)
      status_Aut : Bool;   // STATUS — Simulation is in automatic mode (1 = automatic, 0 = manual)
      status_Man : Bool;   // STATUS — Simulation is in manual mode (1 = manual, 0 = automatic)
      ___________0030_0 { ExternalAccessible := 'False'; ExternalVisible := 'False'; ExternalWritable := 'False'} : Int;
      ___________0030_1 { ExternalAccessible := 'False'; ExternalVisible := 'False'; ExternalWritable := 'False'} : Int;   // ▀▀▀▀ CALCULATED VALUES
      cal_PeakValue : Real;   // CALC — Peak output value
      cal_NatPeriod : Real;   // CALC — Period of natural oscillations (s)
      cal_DampFreq : Real;   // CALC — Damped frequency of the system (rad/s)
      cal_DampFreqHz : Real;   // CALC — Damped frequency of the system (Hz)
      cal_DampPeriod : Real;   // CALC — Period of damped oscillations (s)
      cal_TimeSteady : Real;   // CALC — Time to reach steady state, zero for unstable response (s)
      "cal_Time63%" : Real;   // CALC — Time to reach 63% of steady state (s)
      cal_TimePeak : Real;   // CALC — Time to reach the peak output value (s)
      ___________0040_0 { ExternalAccessible := 'False'; ExternalVisible := 'False'; ExternalWritable := 'False'} : Int;
      ___________0040_1 { ExternalAccessible := 'False'; ExternalVisible := 'False'; ExternalWritable := 'False'} : Int;   // ▀▀▀▀ OPERATING MODE SELECTION
      mode_AutMan : Bool;   // MODE — Automatic/manual mode selection (1 = auto mode, 0 = manual mode)
      mode_ManTime : Real;   // MODE — Manual mode time value (s)
      ___________0050_0 { ExternalAccessible := 'False'; ExternalVisible := 'False'; ExternalWritable := 'False'} : Int;
      ___________0050_1 { ExternalAccessible := 'False'; ExternalVisible := 'False'; ExternalWritable := 'False'} : Int;   // ▀▀▀▀ LIVE TIMING DATA
      actual_Output : Real;   // ACTUAL — SIMULATION OUTPUT VALUE (identical to OUTPUT parameter)
      actual_StartTime : DTL;   // ACTUAL — CPU time when simulation started
      actual_RunTime : Real;   // ACTUAL — Elapsed time since the simulation started (s)
   END_STRUCT;
   // revInfo.REV_BLOCK := 'UT39512';
   // revInfo.REV_NUMBER := '000.102';
   // revInfo.REV_DATE := '2022-02-02';
   // revInfo.REV_AUTHOR := 'M. Gledhill';
END_TYPE

TYPE "UT18151_Dy_SubTimeEventRTC"
TITLE = Dynamic UDT — Subroutine - Event Timer Using RTC
// Event Timer RTC
// stored: IsFailsafeCompliant false
   STRUCT
      revInfo { ExternalWritable := 'False'} : "UT01000_St_SysRevision";   // ▀▀▀▀ UDT CURRENT REVISION
      ___________0010_0 { ExternalAccessible := 'False'; ExternalVisible := 'False'; ExternalWritable := 'False'} : Int;
      ___________0010_1 { ExternalAccessible := 'False'; ExternalVisible := 'False'; ExternalWritable := 'False'} : Int;   // ▀▀▀▀ STATUS SIGNALS
      status_Running { ExternalWritable := 'False'} : Bool;   // STATUS — Event timer is running (1 = running, 0 = stopped)
      ___________0020_0 { ExternalAccessible := 'False'; ExternalVisible := 'False'; ExternalWritable := 'False'} : Int;
      ___________0020_1 { ExternalAccessible := 'False'; ExternalVisible := 'False'; ExternalWritable := 'False'} : Int;   // ▀▀▀▀ EVENT TIMER RESULTS
      actual_StartTime { ExternalWritable := 'False'} : DTL;   // ACTUAL — Start time — RTC value on rising edge of trigger signal
      actual_EndTime { ExternalWritable := 'False'} : DTL;   // ACTUAL — End time — RTC value on falling edge of trigger signal
      actual_Duration { ExternalWritable := 'False'} : LTime;   // ACTUAL — Duration (end time - start time)
      actual_DurationSec { ExternalWritable := 'False'} : Real;   // ACTUAL — Duration (end time - start time) in seconds
   END_STRUCT;
   // revInfo.REV_BLOCK := 'UT18151';
   // revInfo.REV_NUMBER := '000.801';
   // revInfo.REV_DATE := '2021-02-18';
   // revInfo.REV_AUTHOR := 'M. Gledhill';
END_TYPE

TYPE "UT38151_Dy_SubTimeEventRTC"
TITLE = Dynamic UDT [SUBROUTINE] — Event Timer RTC
// PRACTICAL SERIES AUTOMATION LIBRARY (PAL)   —   COPYRIGHT 2020 – M. GLEDHILL (MIT LICENCE)
//                   ———— ◆ ————
// FULL ONLINE DOCUMENTATION IS AVAILABLE AT: https://practicalseries.com/2001-pal/index.html
// stored: IsFailsafeCompliant false
   STRUCT
      revInfo { ExternalWritable := 'False'} : "UT01000_St_SysRevision";   // ▀▀▀▀ UDT CURRENT REVISION
      ___________0010_0 { ExternalAccessible := 'False'; ExternalVisible := 'False'; ExternalWritable := 'False'} : Int;
      ___________0010_1 { ExternalAccessible := 'False'; ExternalVisible := 'False'; ExternalWritable := 'False'} : Int;   // ▀▀▀▀ STATUS SIGNALS
      status_Running { ExternalWritable := 'False'} : Bool;   // STATUS — Event timer is running (1 = running, 0 = stopped)
      ___________0020_0 { ExternalAccessible := 'False'; ExternalVisible := 'False'; ExternalWritable := 'False'} : Int;
      ___________0020_1 { ExternalAccessible := 'False'; ExternalVisible := 'False'; ExternalWritable := 'False'} : Int;   // ▀▀▀▀ EVENT TIMER RESULTS
      actual_StartTime { ExternalWritable := 'False'} : DTL;   // ACTUAL — Start time — RTC value on rising edge of trigger signal
      actual_EndTime { ExternalWritable := 'False'} : DTL;   // ACTUAL — End time — RTC value on falling edge of trigger signal
      actual_Duration { ExternalWritable := 'False'} : LTime;   // ACTUAL — Duration (end time - start time)
      actual_DurationSec { ExternalWritable := 'False'} : Real;   // ACTUAL — Duration (end time - start time) in seconds
   END_STRUCT;
   // revInfo.REV_BLOCK := 'UT38151';
   // revInfo.REV_NUMBER := '002.000';
   // revInfo.REV_DATE := '2022-04-16';
   // revInfo.REV_AUTHOR := 'M. Gledhill';
END_TYPE

